stUserException2.etDiag														:= GD.ET_Diag.ExecutionAborted;
stUserException2.udiDiagExt													:= ET_DiagExt.Exception2FromVis;
stUserException2.sDiagExt													:= FC_EtDiagExtToString(ET_DiagExt.Exception2FromVis);
stUserException2.sMsg														:= 'Test Exception 2 from visualization - TPL.ET_Reaction.SyncStopEL';
stUserException2.udiModuleId												:= vpq_stMachineInterface.i_udiModuleId;
stUserException2.sModuleName												:= vpq_stMachineInterface.i_sModuleName;
stUserException2.etSource													:= TPL.ET_ExceptionSource.Vis;
stUserException2.timDelayTime												:= T#0MS;
stUserException2.wHmiAttributes												:= 0;
stUserException2.xAutoQuit													:= FALSE;
stUserException2.stReaction.axReaction[TPL.ET_Reaction.SyncStopEL]			:= TRUE;

stUserException3.etDiag														:= GD.ET_Diag.ExecutionAborted;
stUserException3.udiDiagExt													:= ET_DiagExt.Exception3FromVis;
stUserException3.sDiagExt													:= FC_EtDiagExtToString(ET_DiagExt.Exception3FromVis);
stUserException3.sMsg														:= 'Test Exception 3 from visualization - TPL.ET_Reaction.SyncStopEH';
stUserException3.udiModuleId												:= vpq_stMachineInterface.i_udiModuleId;
stUserException3.sModuleName												:= vpq_stMachineInterface.i_sModuleName;
stUserException3.etSource													:= TPL.ET_ExceptionSource.Vis;
stUserException3.timDelayTime												:= T#0MS;
stUserException3.wHmiAttributes												:= 0;
stUserException3.xAutoQuit													:= FALSE;
stUserException3.stReaction.axReaction[TPL.ET_Reaction.SyncStopEH]			:= TRUE;

stUserException4.etDiag														:= GD.ET_Diag.ExecutionAborted;
stUserException4.udiDiagExt													:= ET_DiagExt.Exception4FromVis;
stUserException4.sDiagExt													:= FC_EtDiagExtToString(ET_DiagExt.Exception4FromVis);
stUserException4.sMsg														:= 'Test Exception 4 from visualization - TPL.ET_Reaction.StopEndOfCycle';
stUserException4.udiModuleId												:= vpq_stMachineInterface.i_udiModuleId;
stUserException4.sModuleName												:= vpq_stMachineInterface.i_sModuleName;
stUserException4.etSource													:= TPL.ET_ExceptionSource.Vis;
stUserException4.timDelayTime												:= T#0MS;
stUserException4.wHmiAttributes												:= 0;
stUserException4.xAutoQuit													:= FALSE;
stUserException4.stReaction.axReaction[TPL.ET_Reaction.StopEndOfCycle]		:= TRUE;

stUserException5.etDiag														:= GD.ET_Diag.ExecutionAborted;
stUserException5.udiDiagExt													:= ET_DiagExt.Exception5FromVis;
stUserException5.sDiagExt													:= FC_EtDiagExtToString(ET_DiagExt.Exception5FromVis);
stUserException5.sMsg														:= 'Test Exception 5 from visualization - TPL.ET_Reaction.MainsContactorOff';
stUserException5.udiModuleId												:= vpq_stMachineInterface.i_udiModuleId;
stUserException5.sModuleName												:= vpq_stMachineInterface.i_sModuleName;
stUserException5.etSource													:= TPL.ET_ExceptionSource.Vis;
stUserException5.timDelayTime												:= T#0MS;
stUserException5.wHmiAttributes												:= 0;
stUserException5.xAutoQuit													:= FALSE;
stUserException5.stReaction.axReaction[TPL.ET_Reaction.MainsContactorOff]	:= TRUE;
stUserException5.stReaction.axReaction[TPL.ET_Reaction.StopEndOfCycle]		:= TRUE;
END_ACTION

ACTION LoggerVis:
(*For Displaying the LoggerList-Visualization Vis_Logger*)
IF vpiq_udiLogDataListIndexMin < 1 THEN
	vpiq_udiLogDataListIndexMin := 1;
END_IF

IF vpiq_udiLogDataListIndexMin > TPL.Gc_udiMaxNumberOfLogData - 11 THEN
	vpiq_udiLogDataListIndexMin := TPL.Gc_udiMaxNumberOfLogData - 11;
END_IF

FOR udiIndex2 := 1 TO 12 DO
	vpq_astLogDataTableAscii[udiIndex2] := G_stLogDataListAscii.astLogData[vpiq_udiLogDataListIndexMin + udiIndex2 - 1];

	IF G_stLogDataListAscii.astLogData[vpiq_udiLogDataListIndexMin + udiIndex2 - 1].asAsciiData[1]= 'Cmd come' THEN
			vpq_astLogDataTable[udiIndex2].etReason:= TPL. ET_LogDataFilter.CmdCome;
	ELSIF G_stLogDataListAscii.astLogData[vpiq_udiLogDataListIndexMin + udiIndex2 - 1].asAsciiData[1]= 'Cmd go' THEN
			vpq_astLogDataTable[udiIndex2].etReason:= TPL.ET_LogDataFilter.CmdGo;
	ELSIF G_stLogDataListAscii.astLogData[vpiq_udiLogDataListIndexMin + udiIndex2 - 1].asAsciiData[1]= 'StartStep come' THEN
			vpq_astLogDataTable[udiIndex2].etReason:= TPL.ET_LogDataFilter.StartStepCome;
	ELSIF G_stLogDataListAscii.astLogData[vpiq_udiLogDataListIndexMin + udiIndex2 - 1].asAsciiData[1]= 'StartStep go' THEN
			vpq_astLogDataTable[udiIndex2].etReason:= TPL.ET_LogDataFilter.StartStepGo;
	ELSIF G_stLogDataListAscii.astLogData[vpiq_udiLogDataListIndexMin + udiIndex2 - 1].asAsciiData[1]= 'Reaction come' THEN
			vpq_astLogDataTable[udiIndex2].etReason:= TPL.ET_LogDataFilter.ReactionCome;
	ELSIF G_stLogDataListAscii.astLogData[vpiq_udiLogDataListIndexMin + udiIndex2 - 1].asAsciiData[1]= 'Reaction go' THEN
			vpq_astLogDataTable[udiIndex2].etReason:= TPL.ET_LogDataFilter.ReactionGo;
	ELSIF G_stLogDataListAscii.astLogData[vpiq_udiLogDataListIndexMin + udiIndex2 - 1].asAsciiData[1]= 'Exception quit' THEN
			vpq_astLogDataTable[udiIndex2].etReason:= TPL.ET_LogDataFilter.ExceptionQuit;
	ELSIF G_stLogDataListAscii.astLogData[vpiq_udiLogDataListIndexMin + udiIndex2 - 1].asAsciiData[1]= 'Exception come' THEN
			vpq_astLogDataTable[udiIndex2].etReason := TPL.ET_LogDataFilter.ExceptionCome;
	ELSIF G_stLogDataListAscii.astLogData[vpiq_udiLogDataListIndexMin + udiIndex2 - 1].asAsciiData[1]= 'Exception autoquit' THEN
			vpq_astLogDataTable[udiIndex2].etReason:= TPL.ET_LogDataFilter.ExceptionAutoQuit;
	ELSIF G_stLogDataListAscii.astLogData[vpiq_udiLogDataListIndexMin + udiIndex2 - 1].asAsciiData[1]= 'User entry' THEN
			vpq_astLogDataTable[udiIndex2].etReason:= TPL.ET_LogDataFilter.User;
	ELSE
		vpq_astLogDataTable[udiIndex2].etReason:= TPL.ET_LogDataFilter.None;
	END_IF
	vpq_astLogDataTable[udiIndex2].dateDate 		:= STRING_TO_DATE(G_stLogDataListAscii.astLogData[vpiq_udiLogDataListIndexMin + udiIndex2 - 1].asAsciiData[2]);
	vpq_astLogDataTable[udiIndex2].todTime			:= STRING_TO_TOD(G_stLogDataListAscii.astLogData[vpiq_udiLogDataListIndexMin + udiIndex2 - 1].asAsciiData[3]);
	vpq_astLogDataTable[udiIndex2].udiModuleId		:= STRING_TO_UDINT(G_stLogDataListAscii.astLogData[vpiq_udiLogDataListIndexMin + udiIndex2 - 1].asAsciiData[4]);
	vpq_astLogDataTable[udiIndex2].sModuleName		:= G_stLogDataListAscii.astLogData[vpiq_udiLogDataListIndexMin + udiIndex2 - 1].asAsciiData[5];
	vpq_astLogDataTable[udiIndex2].diCMD			:= STRING_TO_DINT(G_stLogDataListAscii.astLogData[vpiq_udiLogDataListIndexMin + udiIndex2 - 1].asAsciiData[6]);
	vpq_astLogDataTable[udiIndex2].diStartStep		:= STRING_TO_DINT(G_stLogDataListAscii.astLogData[vpiq_udiLogDataListIndexMin + udiIndex2 - 1].asAsciiData[7]);

	vpq_astLogDataTable[udiIndex2].etDiag			:= STRING_TO_UDINT(G_stLogDataListAscii.astLogData[vpiq_udiLogDataListIndexMin + udiIndex2 - 1].asAsciiData[8]);
	vpq_astLogDataTable[udiIndex2].udiDiagExt		:= STRING_TO_UDINT(G_stLogDataListAscii.astLogData[vpiq_udiLogDataListIndexMin + udiIndex2 - 1].asAsciiData[10]);
	vpq_astLogDataTable[udiIndex2].sDiagExt			:= G_stLogDataListAscii.astLogData[vpiq_udiLogDataListIndexMin + udiIndex2 - 1].asAsciiData[11];
	vpq_astLogDataTable[udiIndex2].sMsg				:= G_stLogDataListAscii.astLogData[vpiq_udiLogDataListIndexMin + udiIndex2 - 1].asAsciiData[12];
	
	FOR udiIndex3 := 1 TO TPL.Gc_udiMaxNumberOfReactions DO
		IF FIND(G_stLogDataListAscii.astLogData[vpiq_udiLogDataListIndexMin + udiIndex2 - 1].asAsciiData[13], UDINT_TO_STRING(udiIndex3))<>0 THEN
			vpq_astLogDataTable[udiIndex2].stReaction.axReaction[udiIndex3] := TRUE;
		ELSE
			vpq_astLogDataTable[udiIndex2].stReaction.axReaction[udiIndex3] := FALSE;
		END_IF
	END_FOR

	IF    G_stLogDataListAscii.astLogData[vpiq_udiLogDataListIndexMin + udiIndex2 - 1].asAsciiData[14]= '1' THEN
		vpq_astLogDataTable[udiIndex2].etSource:= TPL.ET_ExceptionSource.ModuleController;
	ELSIF G_stLogDataListAscii.astLogData[vpiq_udiLogDataListIndexMin + udiIndex2 - 1].asAsciiData[14]= '2' THEN
		vpq_astLogDataTable[udiIndex2].etSource:= TPL.ET_ExceptionSource.ExceptionHandler;
	ELSIF G_stLogDataListAscii.astLogData[vpiq_udiLogDataListIndexMin + udiIndex2 - 1].asAsciiData[14]= '3' THEN
		vpq_astLogDataTable[udiIndex2].etSource:= TPL.ET_ExceptionSource.Logger;
	ELSIF G_stLogDataListAscii.astLogData[vpiq_udiLogDataListIndexMin + udiIndex2 - 1].asAsciiData[14]= '4' THEN
		vpq_astLogDataTable[udiIndex2].etSource:= TPL.ET_ExceptionSource.Main;
	ELSIF G_stLogDataListAscii.astLogData[vpiq_udiLogDataListIndexMin + udiIndex2 - 1].asAsciiData[14]= '5' THEN
		vpq_astLogDataTable[udiIndex2].etSource:= TPL.ET_ExceptionSource.Vis;
	ELSIF G_stLogDataListAscii.astLogData[vpiq_udiLogDataListIndexMin + udiIndex2 - 1].asAsciiData[14]= '6' THEN
		vpq_astLogDataTable[udiIndex2].etSource:= TPL.ET_ExceptionSource.User;
	ELSIF G_stLogDataListAscii.astLogData[vpiq_udiLogDataListIndexMin + udiIndex2 - 1].asAsciiData[14]= '7' THEN
		vpq_astLogDataTable[udiIndex2].etSource:= TPL.ET_ExceptionSource.NodeModule;
	ELSIF G_stLogDataListAscii.astLogData[vpiq_udiLogDataListIndexMin + udiIndex2 - 1].asAsciiData[14]= '8' THEN
		vpq_astLogDataTable[udiIndex2].etSource:= TPL.ET_ExceptionSource.AxisModule;
	ELSIF G_stLogDataListAscii.astLogData[vpiq_udiLogDataListIndexMin + udiIndex2 - 1].asAsciiData[14]= '9' THEN
		vpq_astLogDataTable[udiIndex2].etSource:= TPL.ET_ExceptionSource.MultiBeltModule;
	ELSIF G_stLogDataListAscii.astLogData[vpiq_udiLogDataListIndexMin + udiIndex2 - 1].asAsciiData[14]= '10' THEN
		vpq_astLogDataTable[udiIndex2].etSource:= TPL.ET_ExceptionSource.SmartInfeedModule;
	ELSIF G_stLogDataListAscii.astLogData[vpiq_udiLogDataListIndexMin + udiIndex2 - 1].asAsciiData[14]= '11' THEN
		vpq_astLogDataTable[udiIndex2].etSource:= TPL.ET_ExceptionSource.RoboticModule;
	ELSIF G_stLogDataListAscii.astLogData[vpiq_udiLogDataListIndexMin + udiIndex2 - 1].asAsciiData[14]= '12' THEN
		vpq_astLogDataTable[udiIndex2].etSource:= TPL.ET_ExceptionSource.UnwinderModule;
	ELSIF G_stLogDataListAscii.astLogData[vpiq_udiLogDataListIndexMin + udiIndex2 - 1].asAsciiData[14]= '13' THEN
		vpq_astLogDataTable[udiIndex2].etSource:= TPL.ET_ExceptionSource.SealingModule;
	ELSIF G_stLogDataListAscii.astLogData[vpiq_udiLogDataListIndexMin + udiIndex2 - 1].asAsciiData[14]= '14' THEN
		vpq_astLogDataTable[udiIndex2].etSource:= TPL.ET_ExceptionSource.AtvModule;
	ELSIF G_stLogDataListAscii.astLogData[vpiq_udiLogDataListIndexMin + udiIndex2 - 1].asAsciiData[14]= '15' THEN
		vpq_astLogDataTable[udiIndex2].etSource:= TPL.ET_ExceptionSource.IlxModule;
	ELSIF G_stLogDataListAscii.astLogData[vpiq_udiLogDataListIndexMin + udiIndex2 - 1].asAsciiData[14]= '16' THEN
		vpq_astLogDataTable[udiIndex2].etSource:= TPL.ET_ExceptionSource.CrankModule;
	ELSIF G_stLogDataListAscii.astLogData[vpiq_udiLogDataListIndexMin + udiIndex2 - 1].asAsciiData[14]= '17' THEN
		vpq_astLogDataTable[udiIndex2].etSource:= TPL.ET_ExceptionSource.ValveModule;
	ELSIF G_stLogDataListAscii.astLogData[vpiq_udiLogDataListIndexMin + udiIndex2 - 1].asAsciiData[14]= '18' THEN
		vpq_astLogDataTable[udiIndex2].etSource:= TPL.ET_ExceptionSource.CapperModule;
	ELSE
		vpq_astLogDataTable[udiIndex2].etSource:= TPL.ET_ExceptionSource.None;
	END_IF
	
	vpq_astLogDataTable[udiIndex2].xAutoQuit	:= STRING_TO_BOOL(G_stLogDataListAscii.astLogData[vpiq_udiLogDataListIndexMin + udiIndex2 - 1].asAsciiData[15]);
END_FOR


vpq_udiLogDataListIndexMax := vpiq_udiLogDataListIndexMin + 11;

vpiq_udiNumberOfLogData := G_stLogDataListAscii.udiNumberOfLogData;
IF vpq_udiLogDataListIndexMax > G_stLogDataListAscii.udiNumberOfLogData - 1  THEN
	vpq_xLogDataScrollDown := TRUE;

ELSE
	vpq_xLogDataScrollDown := FALSE;
END_IF

IF vpiq_xButtonLogDataListDetails AND NOT vpq_xShowLogDataListDetails THEN
	vpq_xShowLogDataListDetails				:= TRUE;
	vpiq_xButtonLogDataListDetails			:= FALSE;
ELSIF vpiq_xButtonLogDataListDetails AND vpq_xShowLogDataListDetails THEN
	vpq_xShowLogDataListDetails				:= FALSE;
	vpiq_xButtonLogDataListDetails			:= FALSE;
END_IF
END_ACTION

ACTION MainPageCmdTable:
(* Find the current table*)
vpq_udiNumberOfCmdStepsModule		:= 0; (* Default values, for security *)
pstEQCMDTableListEntry	:= 0;
pstEQCMDTable			:= 0;

IF(vpq_stMachineInterface.q_diCmdActive <> 0 AND vpq_stMachineInterface.iq_stExt.udiNumberOfCmdTables > 0 AND vpq_stMachineInterface.iq_stExt.pstListofCMDTables <> 0) THEN
	FOR udiTmp2 := 1 TO vpq_stMachineInterface.iq_stExt.udiNumberOfCMDTables DO
		pstEQCMDTableListEntry := vpq_stMachineInterface.iq_stExt.pstListofCMDTables +  UDINT_TO_DWORD((udiTmp2-1)*SIZEOF(pstEQCMDTableListEntry^));
		IF(pstEQCMDTableListEntry^.diCMD = vpq_stMachineInterface.q_diCmdActive) THEN (* Found *)
			vpq_udiNumberOfCmdStepsModule := pstEQCMDTableListEntry^.udiNumberOfCmdSteps;
			vpq_udiNumberOfCmdStepsMain := vpq_udiNumberOfCmdStepsModule;
			pstEQCMDTable := pstEQCMDTableListEntry^.pstCMDTable;
			vpq_sCmdTitelMain := pstEQCMDTableListEntry^.sTitle;
			EXIT;
		END_IF
	END_FOR
END_IF

(***********************************************************************************************************************)
(* Check the limits of the Vis/ shown table *)
udiIndexOldMainTable := 0;
IF vpiq_udiIndexMinMain <> udiIndexOldMainTable THEN
														(*More than 10 steps ??*)
	IF (vpiq_udiIndexMinMain + 9 < vpq_udiNumberOfCmdStepsMain) THEN
		udiIndexMaxMainTable := vpiq_udiIndexMinMain + 9;
	ELSE
		udiIndexMaxMainTable := vpq_udiNumberOfCmdStepsMain;
	END_IF
														(*Additional safety check*)
	IF (vpiq_udiIndexMinMain < 1) OR (vpiq_udiIndexMinMain > vpq_udiNumberOfCmdStepsMain) THEN
		vpiq_udiIndexMinMain :=1;
		udiIndexMaxMainTable := 10;
	END_IF

	udiIndexOldMainTable := vpiq_udiIndexMinMain;
END_IF (*udiEQMainTableIndexMin <> udiEQMainTableIndexOld*)

vpq_xDisableScrollUpMain	:= NOT (vpiq_udiIndexMinMain > 1);
vpq_xDisableScrollDownMain	:= NOT (vpiq_udiIndexMinMain + 9 < vpq_udiNumberOfCmdStepsMain) ;

(***********************************************************************************************************************)
(*Refresh the values in the table if more then "Max commands" should be shown!*)
IF(pstEQCMDTable <> 0) THEN
	FOR udiCounter := udiIndexOldMainTable TO udiIndexMaxMainTable DO
		pstEQCMDTableEntry := pstEQCMDTable +  UDINT_TO_DWORD(((udiCounter-1) * SIZEOF(pstEQCMDTable^)));
		vpq_astActualCmdTableMain[udiCounter - udiIndexOldMainTable + 1] := pstEQCMDTableEntry^;
	END_FOR
	FOR udiCounter := udiIndexMaxMainTable + 1 TO udiIndexOldMainTable + 9 DO
		vpq_astActualCmdTableMain[udiCounter - udiIndexOldMainTable + 1] := c_stEmptyCmdTableStep;
	END_FOR
END_IF
END_ACTION

ACTION ModuleNavigationIn:
(* Navigation *)

(* 2D navigation *)
IF(vpiq_xNavUp OR vpiq_xNavDown OR vpiq_xNavLeft OR vpiq_xNavRight) THEN
	IF vpiq_xNavRight THEN
		(* Move the the next module on the same level *)
		IF audiHierarchy[udiCurrentLevel] + 1 <= udiCurrentLevelSize + udiCurrentNumberOfControlModules  THEN
			audiHierarchy[udiCurrentLevel] := audiHierarchy[udiCurrentLevel] + 1;
			IF audiHierarchy[udiCurrentLevel]  > udiCurrentLevelSize THEN
				udiControlModuleSelectedInLevel	:= udiCurrentLevel;
				vpq_udiActiveControlModuleNumber:= audiHierarchy[udiCurrentLevel]-udiCurrentLevelSize;
			END_IF
		END_IF
	END_IF
	IF vpiq_xNavLeft THEN
		(* Move the the previous module on the same level *)
		IF audiHierarchy[udiCurrentLevel] -1 >= 1 THEN
			audiHierarchy[udiCurrentLevel] := audiHierarchy[udiCurrentLevel] - 1;
			vpq_udiActiveControlModuleNumber:= audiHierarchy[udiCurrentLevel]-udiCurrentLevelSize;
			IF audiHierarchy[udiCurrentLevel] <= udiCurrentLevelSize THEN
				udiControlModuleSelectedInLevel	:= 0;
				vpq_udiActiveControlModuleNumber:= 0;
			END_IF
		END_IF (* ELSE ignore *)
	END_IF
	IF vpiq_xNavUp THEN
		(* Move one level up *)
		udiControlModuleSelectedInLevel := 0;
		vpq_udiActiveControlModuleNumber:= 0;
		IF udiCurrentLevel - 1 >= 1 THEN
			udiCurrentLevel := udiCurrentLevel - 1;
		END_IF (* ELSE ignore *)
	END_IF
	IF vpiq_xNavDown THEN
		(* Move one level down *)
		IF (udiCurrentLevel + 1 <= c_udiMaxHierarchyLevels) AND (xCurrentHasSubModules OR xCurrentHasControlModules) THEN
			udiCurrentLevel := udiCurrentLevel + 1;
			audiHierarchy[udiCurrentLevel] := 1;
			IF NOT xCurrentHasSubModules AND xCurrentHasControlModules THEN
				udiControlModuleSelectedInLevel := udiCurrentLevel;
				vpq_udiActiveControlModuleNumber:= audiHierarchy[udiCurrentLevel];
			ELSE
				udiControlModuleSelectedInLevel	:= 0;
				vpq_udiActiveControlModuleNumber:= 0;
			END_IF

		END_IF (* ELSE ignore *)
	END_IF

	vpiq_xNavUp		:= FALSE;
	vpiq_xNavDown	:= FALSE;
	vpiq_xNavLeft	:= FALSE;
	vpiq_xNavRight	:= FALSE;
	
	xUpdateData := TRUE;
END_IF (* End 2D navbutton hit *)

(* Direct navigation (on level 2 and 3) *)
(* Module level *)
IF vpiq_axModuleList[1] OR vpiq_axModuleList[2] OR vpiq_axModuleList[3] OR vpiq_axModuleList[4] OR vpiq_axModuleList[5] OR
   vpiq_axControlModuleList[1] OR vpiq_axControlModuleList[2] OR vpiq_axControlModuleList[3] OR vpiq_axControlModuleList[4] OR vpiq_axControlModuleList[5] THEN
	udiCurrentLevel := 2;
	udiCurrentLevel := 2;
	FOR udiTmp := 1 TO 5 DO
		(*select an equipment module via the buttons on level 2*)
		IF(vpiq_axModuleList[udiTmp]) THEN
			audiHierarchy[udiCurrentLevel] := udiTmp + udiMinModuleList - 1;
			vpiq_axModuleList[udiTmp] := FALSE;
			udiControlModuleSelectedInLevel := 0;
			vpq_udiActiveControlModuleNumber:= 0;
		END_IF
		(*select a control module via the buttons on level 2*)
		IF vpiq_axControlModuleList[udiTmp] THEN
			audiHierarchy[udiCurrentLevel] := udiTmp + udiMinModuleList - 1;
			udiControlModuleSelectedInLevel	:= udiCurrentLevel;
			vpiq_axControlModuleList[udiTmp] := FALSE;
		END_IF
	END_FOR
	xUpdateData := TRUE;
END_IF
IF vpiq_xModuleListDown THEN
	vpiq_xModuleListDown := FALSE;
	IF(udiMinModuleList > 1) THEN
		udiMinModuleList := udiMinModuleList - 1;
	END_IF
	xUpdateData := TRUE;
END_IF
IF vpiq_xModuleListUp THEN
	vpiq_xModuleListUp := FALSE;
	IF(udiMinModuleList + 4 <= vpq_stMachineInterface.iq_stExt.udiNumberOfSubModules + vpq_stMachineInterface.iq_stExt.udiNumberOfControlModules) THEN
		udiMinModuleList := udiMinModuleList + 1;
	END_IF
	xUpdateData := TRUE;
END_IF
(* Submodule level *)
IF(udiCurrentLevel >= 2) THEN (* Impossible if the main machine is selected *)
	IF vpiq_axSubModuleList[1] OR vpiq_axSubModuleList[2] OR vpiq_axSubModuleList[3] OR vpiq_axSubModuleList[4] OR vpiq_axSubModuleList[5] OR
	   vpiq_axSubControlModuleList[1] OR vpiq_axSubControlModuleList[2] OR vpiq_axSubControlModuleList[3] OR vpiq_axSubControlModuleList[4] OR vpiq_axSubControlModuleList[5] THEN
		udiCurrentLevel := 3;
		FOR udiTmp := 1 TO 5 DO
			(*select an equipment module via the buttons on level 3*)
			IF(vpiq_axSubModuleList[udiTmp]) THEN
				audiHierarchy[udiCurrentLevel] := udiTmp + udiMinSubModuleList - 1;
				vpiq_axSubModuleList[udiTmp] := FALSE;
				udiControlModuleSelectedInLevel	:= 0;
				vpq_udiActiveControlModuleNumber	:= 0;
			END_IF
			(*select a control module via the buttons on level 3*)
			IF vpiq_axSubControlModuleList[udiTmp] THEN
				audiHierarchy[udiCurrentLevel] := udiTmp + udiMinSubModuleList - 1;
				vpiq_axSubControlModuleList[udiTmp] := FALSE;
				udiControlModuleSelectedInLevel	:= udiCurrentLevel;
			END_IF
		END_FOR
		xUpdateData := TRUE;
	END_IF
	IF vpiq_xSubModuleListDown THEN
		vpiq_xSubModuleListDown := FALSE;
		IF(udiMinSubModuleList > 1) THEN
			udiMinSubModuleList := udiMinSubModuleList - 1;
		END_IF
		xUpdateData := TRUE;
	END_IF
	IF vpiq_xSubModuleListUp THEN
		vpiq_xSubModuleListUp := FALSE;
		IF(udiMinSubModuleList + 4 < udiCurrentLevel3Size + udiNumberOfControlModulesLevel2) THEN
			udiMinSubModuleList := udiMinSubModuleList + 1;
		END_IF
		xUpdateData := TRUE;
	END_IF
END_IF
END_ACTION

ACTION ModuleNavigationOut:
(* update 2d nav data *)
vpq_sNameNavUp		:= '';
vpq_sNameNavRight	:= '';
vpq_sNameNavLeft		:= '';

IF pstCurrentParent = 0 THEN
	udiCurrentLevelSize := 1;
ELSE
	udiCurrentLevelSize := pstCurrentParent^.iq_stExt.udiNumberOfSubModules;

	vpq_sNameNavUp := pstCurrentParent^.i_sModuleName;
	(*If next module is a equipment module*)
	IF (audiHierarchy[udiCurrentLevel] + 1 <= udiCurrentLevelSize) THEN
		pstTmp := pstCurrentParent^.iq_stExt.dwSubModulesItf
			+ UDINT_TO_DWORD((audiHierarchy[udiCurrentLevel] -1 + 1) * SIZEOF(vpq_stCurrentModuleStandardInterface));
		vpq_sNameNavRight := pstTmp^.i_sModuleName;
	(*If next module is a control module*)
	ELSIF audiHierarchy[udiCurrentLevel] + 1 <= udiCurrentLevelSize + pstCurrentParent^.iq_stExt.udiNumberOfControlModules THEN
		pstControlModuleInterface	:= pstCurrentParent^.iq_stExt.dwControlModulesItf + UDINT_TO_DWORD((audiHierarchy[udiCurrentLevel]-udiCurrentLevelSize) * SIZEOF(pstControlModuleInterface^));
		vpq_sNameNavRight			:= pstControlModuleInterface^.sControlModuleName;
	END_IF
	IF (audiHierarchy[udiCurrentLevel] -1 >= 1) THEN
		(*If former module is a equipment module*)
		IF audiHierarchy[udiCurrentLevel]-1 <= udiCurrentLevelSize THEN
			pstTmp := pstCurrentParent^.iq_stExt.dwSubModulesItf
				+ UDINT_TO_DWORD((audiHierarchy[udiCurrentLevel] -1 - 1) * SIZEOF(vpq_stCurrentModuleStandardInterface));
			vpq_sNameNavLeft := pstTmp^.i_sModuleName;
		(*If former module is a control module*)
		ELSE
			pstControlModuleInterface	:= pstCurrentParent^.iq_stExt.dwControlModulesItf + UDINT_TO_DWORD((audiHierarchy[udiCurrentLevel]-udiCurrentLevelSize-2) * SIZEOF(pstControlModuleInterface^));
			vpq_sNameNavLeft				:= pstControlModuleInterface^.sControlModuleName;
		END_IF
	END_IF
END_IF

xCurrentHasControlModules := pstCurrent^.iq_stExt.udiNumberOfControlModules > 0;
xCurrentHasSubModules := ((pstCurrent^.iq_stExt.udiNumberOfSubModules > 0) AND udiControlModuleSelectedInLevel = 0);
xCurrentIsNoNodeModule := (pstCurrent^.q_dwModuleType <>  UDINT_TO_DWORD(TPL.ET_ModuleType.NodeModule));
IF((xCurrentIsNoNodeModule OR xCurrentHasControlModules) AND udiControlModuleSelectedInLevel = 0) THEN
	IF(pstCurrentParent <> 0) THEN (* Security check *)
		pdwTmp := ADR(pstCurrentParent^.iq_stExt.pdwSubModulesAddItf^)
			+  UDINT_TO_DWORD((audiHierarchy[udiCurrentLevel] - 1) * SIZEOF(dwDummy));
		dwCurrentAddInterface := pdwTmp^;
	END_IF
END_IF

vpq_xEnableNavUp		:= (udiCurrentLevel - 1 >= 1);
vpq_xEnableNavDown	:= (udiCurrentLevel < c_udiMaxHierarchyLevels) AND (xCurrentHasSubModules OR xCurrentHasControlModules) AND udiControlModuleSelectedInLevel = 0 ;
vpq_xEnableNavLeft	:= (audiHierarchy[udiCurrentLevel] -1 >= 1);
vpq_xEnableNavRight	:= (audiHierarchy[udiCurrentLevel] + 1 <= udiCurrentLevelSize + udiCurrentNumberOfControlModules)AND(udiCurrentLevel >=2);

IF vpq_xEnableNavDown THEN
	(* Name of the first submodule of the current module *)
	IF xCurrentHasSubModules THEN
		pstTmp := pstCurrent^.iq_stExt.dwSubModulesItf;
		vpq_sNameNavDown := pstTmp^.i_sModuleName;
	ELSE
		pstControlModuleInterface	:= pstCurrent^.iq_stExt.dwControlModulesItf;
		vpq_sNameNavDown				:= pstControlModuleInterface^.sControlModuleName;
	END_IF

ELSE
	vpq_sNameNavDown := '';
END_IF

(* Update direct nav data *)
(* Module level *)
vpq_xDisableModuleListDown	:= NOT (udiMinModuleList > 1);
vpq_xDisableModuleListUp		:= NOT (udiMinModuleList + 5 <= vpq_stMachineInterface.iq_stExt.udiNumberOfSubModules + vpq_stMachineInterface.iq_stExt.udiNumberOfControlModules);
FOR udiTmp := 1 TO 5 DO
	vpq_axControlModuleValid[udiTmp]:=FALSE;
	audiControlModuleNumber[udiTmp]:= 0 (*-1*);
	vpq_asToolTipControlModuleList[udiTmp] := 'None';
	vpq_axDisableModuleList[udiTmp] := NOT ((udiTmp - 1 + udiMinModuleList) <= vpq_stMachineInterface.iq_stExt.udiNumberOfSubModules);
	vpq_axActiveModuleList[udiTmp] := (udiCurrentLevel >= 2) AND (audiHierarchy[2] = (udiTmp - 1 + udiMinModuleList));
	vpq_axControlModuleActive[udiTmp] := FALSE;
	(*Show button for equipment module*)
	IF(NOT vpq_axDisableModuleList[udiTmp]) THEN
		pstTmp := vpq_stMachineInterface.iq_stExt.dwSubModulesItf
			+ UDINT_TO_DWORD(((udiTmp - 1 + udiMinModuleList) - 1) * SIZEOF(vpq_stCurrentModuleStandardInterface));
		vpq_audiIdModuleList[udiTmp] := pstTmp^.i_udiModuleId;
		vpq_axIdModuleListValid[udiTmp] := TRUE;
		
		vpq_asNameModuleList[udiTmp] := pstTmp^.i_sModuleName;
	(*Show button for control module*)
	ELSE
		vpq_audiIdModuleList[udiTmp] := 0 (*-1*);
		vpq_axIdModuleListValid[udiTmp] := FALSE;
		vpq_asNameModuleList[udiTmp] := 'None';
		IF vpq_stMachineInterface.iq_stExt.udiNumberOfControlModules <> 0 AND udiTmp <= vpq_stMachineInterface.iq_stExt.udiNumberOfControlModules + vpq_stMachineInterface.iq_stExt.udiNumberOfSubModules THEN
			pstControlModuleInterface	:= vpq_stMachineInterface.iq_stExt.dwControlModulesItf + UDINT_TO_DWORD((udiTmp - vpq_stMachineInterface.iq_stExt.udiNumberOfSubModules - 1 + udiMinModuleList)-1) * SIZEOF(pstControlModuleInterface^);
			vpq_asToolTipControlModuleList[udiTmp]:= pstControlModuleInterface^.sControlModuleName;
			vpq_axControlModuleActive[udiTmp] := (udiCurrentLevel >= 2) AND (audiHierarchy[2] = (udiTmp - 1 + udiMinModuleList));
			vpq_axControlModuleValid[udiTmp]:=TRUE;
			audiControlModuleNumber[udiTmp]:= pstControlModuleInterface^.udiControlModuleNumber;
			vpq_asControlModuleButtonName[udiTmp]:= CONCAT(STR1:='Type: ',STR2:= CONCAT(STR1:= UDINT_TO_STRING(pstControlModuleInterface^.udiControlModuleType), STR2:= CONCAT(STR1:='   #: ',STR2:= UDINT_TO_STRING(pstControlModuleInterface^.udiControlModuleNumber))));
		END_IF
	END_IF
END_FOR

(* Submodule level *)
IF (udiMinSubModuleList + 4 > udiCurrentLevel3Size+udiNumberOfControlModulesLevel2) THEN
	udiMinSubModuleList := 1;
END_IF
vpq_xDisableSubModuleListDown	:= NOT (udiMinSubModuleList > 1);
vpq_xDisableSubModuleListUp		:= NOT (udiMinSubModuleList + 5 <= udiCurrentLevel3Size+udiNumberOfControlModulesLevel2)AND NOT (udiCurrentLevel = 2 AND xControlModuleSelected);
FOR udiTmp := 1 TO 5 DO
	vpq_axDisableSubModuleList[udiTmp] := NOT ((udiTmp - 1 + udiMinSubModuleList) <= udiCurrentLevel3Size);
	vpq_axActiveSubModuleList[udiTmp] := (udiCurrentLevel >= 3) AND (audiHierarchy[3] = (udiTmp - 1 + udiMinSubModuleList));
	vpq_audiIdSubModuleList[udiTmp] := 0 (*-1*);
	vpq_axIdSubModuleListValid[udiTmp] := FALSE;
	vpq_asNameSubModuleList[udiTmp] := 'None';
	vpq_axSubControlModuleValid[udiTmp]:= FALSE;
	audiSubControlModuleID[udiTmp]:= 0 (*-1*);
	vpq_asToolTipSubControlModuleList[udiTmp] := 'None';
	vpq_axSubControlModuleActive[udiTmp] := FALSE;
	(*Show button for equipment module*)
	IF(NOT vpq_axDisableSubModuleList[udiTmp]) THEN
		IF(pstCurrentFirstLevel3Module <> 0) THEN
			pstTmp := ADR(pstCurrentFirstLevel3Module^)
				+  UDINT_TO_DWORD(((udiTmp - 1 + udiMinSubModuleList) - 1) * SIZEOF(vpq_stCurrentModuleStandardInterface));
			vpq_audiIdSubModuleList[udiTmp] := pstTmp^.i_udiModuleId;
			vpq_axIdSubModuleListValid[udiTmp] := TRUE;
			
			vpq_asNameSubModuleList[udiTmp] := pstTmp^.i_sModuleName;
		END_IF
	(*Show button for control module*)
	ELSE
		IF udiCurrentLevel >= 2 AND udiControlModuleSelectedInLevel <> 2 THEN
			IF pstCurrentLevel2 <> 0 THEN
				IF pstCurrentLevel2^.iq_stExt.udiNumberOfControlModules <> 0 AND udiTmp <= pstCurrentLevel2^.iq_stExt.udiNumberOfControlModules + udiCurrentLevel3Size THEN
					pstControlModuleInterface	:= pstCurrentLevel2^.iq_stExt.dwControlModulesItf + UDINT_TO_DWORD((udiTmp - pstCurrentLevel2^.iq_stExt.udiNumberOfSubModules - 1 + udiMinSubModuleList - 1) * SIZEOF(pstControlModuleInterface^));
					vpq_asToolTipSubControlModuleList[udiTmp]:= pstControlModuleInterface^.sControlModuleName;
					vpq_asSubControlModuleButtonName[udiTmp]:= CONCAT(STR1:='Type: ',STR2:= CONCAT(STR1:= UDINT_TO_STRING(pstControlModuleInterface^.udiControlModuleType), STR2:= CONCAT(STR1:='   #: ',STR2:= UDINT_TO_STRING(pstControlModuleInterface^.udiControlModuleNumber))));
					vpq_axSubControlModuleActive[udiTmp] :=  (udiCurrentLevel >= 3) AND (audiHierarchy[3] = (udiTmp - 1 + udiMinSubModuleList));
					vpq_axSubControlModuleValid[udiTmp]:= TRUE;
					audiSubControlModuleID[udiTmp]:= pstControlModuleInterface^.udiControlModuleNumber;
				END_IF
			END_IF
		END_IF
	END_IF
END_FOR

// iEQTableIndexMin := 1;
//iEQTableIndexOld := 0;

(*Select current control module*)
FOR udiTmp := 1 TO 5 DO
	IF vpq_axControlModuleActive[udiTmp] THEN
		vpq_udiActiveControlModuleNumber:= audiControlModuleNumber[udiTmp];
	END_IF
	IF vpq_axSubControlModuleActive[udiTmp] THEN
		vpq_udiActiveControlModuleNumber:= audiSubControlModuleID[udiTmp];
	END_IF
END_FOR
END_ACTION

ACTION ModuleReaction:
stModuleReactions		:=pstCurrent^.i_stReaction;

IF vpiq_xModuleReactionUp THEN
	vpq_udiModuleReactionIndexMin := vpq_udiModuleReactionIndexMin + 1;
	vpiq_xModuleReactionUp := FALSE;
ELSIF vpiq_xModuleReactionDown THEN
	vpq_udiModuleReactionIndexMin := vpq_udiModuleReactionIndexMin - 1;
	vpiq_xModuleReactionDown := FALSE;
END_IF

IF vpq_udiModuleReactionIndexMin <> udiModuleReactionIndexOld THEN
														(*More than 10 steps ??*)
	IF (vpq_udiModuleReactionIndexMin + 9 < TPL.Gc_udiMaxNumberOfReactions) THEN
		udiModuleReactionIndexMax := vpq_udiModuleReactionIndexMin + 9;
	ELSE
		udiModuleReactionIndexMax := TPL.Gc_udiMaxNumberOfReactions;
	END_IF
														(*Additional safety check*)
	IF (vpq_udiModuleReactionIndexMin < 1) THEN
		vpq_udiModuleReactionIndexMin :=1;
		udiModuleReactionIndexMax := 10;
 	ELSIF (vpq_udiModuleReactionIndexMin > TPL.Gc_udiMaxNumberOfReactions-9)THEN
		vpq_udiModuleReactionIndexMin :=TPL.Gc_udiMaxNumberOfReactions-9;
		udiModuleReactionIndexMax := 10;
	END_IF

	udiModuleReactionIndexOld := vpq_udiModuleReactionIndexMin;
END_IF

IF TPL.Gc_udiMaxNumberOfReactions<10 THEN
	udiMaxValue := TPL.Gc_udiMaxNumberOfReactions;
ELSE
	udiMaxValue := 10;
END_IF

FOR udiCount2 := 1 TO udiMaxValue  DO
	vpq_axModuleReaction[udiCount2] := stModuleReactions.axReaction[vpq_udiModuleReactionIndexMin + udiCount2 - 1];
END_FOR
END_ACTION

ACTION ModuleVisController:
(* Begin of area for vis control fbs of different module types *)
(* SetCurrentModule(); has to be called after each special vis-controller, because it could have requested to change the current module via diSetAsCurrentModule *)

vpiq_fbAxisModuleVisController(	i_xEnable				:= vpq_xDoEnable, 
								i_pstMachineStandardItf	:= ADR(SR_MainMachine.stMachineInterface),
								i_pstCurrentStandardItf	:= pstCurrent, 
								i_dwCurrentAddItf		:= dwCurrentAddInterface, 
								i_xUpdateData			:= xUpdateForOtherFBs,
								i_udiCurrentJogTarget	:= G_udiManualModuleSelect, 
								iq_stExceptionList		:= G_stExceptionList,
								iq_stLogDataList		:= G_stLogDataList,
								q_xActive				=> , 
								q_xReady				=> , 
								q_etDiag				=> , 
								q_etDiagExt				=> , 
								q_sMsg					=> , 
								q_udiSetAsCurrentModule	=> udiSetAsCurrentModule,
								q_udiSetAsJogTarget		=> udiSetAsJogTarget);
SetCurrentModule();

(* Example 
vpiq_fbExampleLeafModuleVisController(	i_xEnable				:= vpq_xDoEnable, 
										i_pstMachineStandardItf	:= ADR(SR_MainMachine.stMachineInterface), 
										i_pstCurrentStandardItf	:= pstCurrent, 
										i_dwCurrentAddItf		:= dwCurrentAddInterface, 
										i_xUpdateData			:= xUpdateForOtherFBs, 
										i_udiCurrentJogTarget	:= G_udiManualModuleSelect, 
										iq_stExceptionList		:= G_stExceptionList,
										iq_stLogDataList		:= G_stLogDataList, 
										q_xActive				=> , 
										q_xReady				=> , 
										q_etDiag				=> , 
										q_etDiagExt				=> , 
										q_sMsg					=> , 
										q_udiSetAsCurrentModule	=> udiSetAsCurrentModule, 
										q_udiSetAsJogTarget		=> udiSetAsJogTarget);
SetCurrentModule();
*)

(* RoboticModule *)
(*vpiq_fbRoboticModuleVisController(	i_xEnable				:= vpq_xDoEnable, 
									i_pstMachineStandardItf	:= ADR(SR_MainMachine.stMachineInterface),
									i_pstCurrentStandardItf	:= pstCurrent, 
									i_dwCurrentAddItf		:= dwCurrentAddInterface, 
									i_xUpdateData			:= xUpdateForOtherFBs,
									i_udiCurrentJogTarget	:= G_udiManualModuleSelect, 
									iq_stExceptionList		:= G_stExceptionList,
									iq_stLogDataList		:= G_stLogDataList,
									q_xActive				=> , 
									q_xReady				=> , 
									q_etDiag				=> , 
									q_etDiagExt				=> , 
									q_sMsg					=> , 
									q_udiSetAsCurrentModule	=> udiSetAsCurrentModule,
									q_udiSetAsJogTarget		=> udiSetAsJogTarget);
SetCurrentModule();*)
END_ACTION

ACTION OpModeControl:
IFB_RTOPMode(CLK:= G_xDoPrepare OR G_xDoAuto OR G_xDoManual OR G_xDoJogMachine OR G_xDoBrakeRelease OR G_xDoTestMulticarrier OR G_xDoTrackCalibration);
IF G_xDoPrepare THEN
	IF g_xPrepareActive AND G_xPrepareEpas AND IFB_RTOPMode.Q THEN
		g_xPrepareActive := FALSE;
		G_xPrepareEpas:= FALSE;
	ELSIF IFB_RTOPMode.Q THEN
		g_xPrepareActive := TRUE;
		G_xPrepareEpas:= TRUE;
	END_IF
	G_xTestMulticarrierEpas := FALSE;
	G_xAutoEpas := FALSE;
	G_xManualEpas := FALSE;
	G_xJogMachineEpas := FALSE;
	G_xBrakeReleaseEpas := FALSE;
	G_xTrackCalibrationEpas := FALSE;

ELSIF G_xDoAuto THEN
	IF G_xAutoActive AND G_xAutoEpas AND IFB_RTOPMode.Q THEN
		G_xAutoActive := FALSE;
		G_xAutoEpas := FALSE;
	ELSIF IFB_RTOPMode.Q THEN
		G_xAutoActive := TRUE;
		G_xAutoEpas := TRUE;
	END_IF
	G_xTestMulticarrierEpas := FALSE;
	G_xManualEpas := FALSE;
	G_xJogMachineEpas := FALSE;
	G_xBrakeReleaseEpas := FALSE;
	G_xPrepareEpas:= FALSE;
	G_xTrackCalibrationEpas := FALSE;

ELSIF G_xDoManual THEN
	IF G_xManualActive AND G_xManualEpas AND IFB_RTOPMode.Q THEN
		G_xManualActive := FALSE;
		G_xManualEpas := FALSE;
	ELSIF IFB_RTOPMode.Q THEN
		g_xManualActive := TRUE;
		G_xManualEpas := TRUE;
	END_IF
	G_xTestMulticarrierEpas := FALSE;
	G_xJogMachineEpas := FALSE;
	G_xBrakeReleaseEpas := FALSE;
	G_xPrepareEpas:= FALSE;
	G_xAutoEpas := FALSE;
	G_xTrackCalibrationEpas := FALSE;

ELSIF g_xDoJogMachine THEN
	IF g_xJogMachineActive AND G_xJogMachineEpas AND IFB_RTOPMode.Q THEN
		g_xJogMachineActive := FALSE;
		G_xJogMachineEpas := FALSE;
	ELSIF IFB_RTOPMode.Q THEN
		g_xJogMachineActive := TRUE;
		G_xJogMachineEpas := TRUE;
	END_IF
	G_xTestMulticarrierEpas := FALSE;
	G_xBrakeReleaseEpas := FALSE;
	G_xPrepareEpas:= FALSE;
	G_xAutoEpas := FALSE;
	G_xManualEpas := FALSE;
	G_xTrackCalibrationEpas := FALSE;

ELSIF g_xDoBrakeRelease THEN
	IF g_xBrakeReleaseActive AND G_xBrakeReleaseEpas AND IFB_RTOPMode.Q THEN
		g_xBrakeReleaseActive := FALSE;
		G_xBrakeReleaseEpas := FALSE;
	ELSIF IFB_RTOPMode.Q THEN
		g_xBrakeReleaseActive := TRUE;
		G_xBrakeReleaseEpas := TRUE;
	END_IF
	G_xTestMulticarrierEpas := FALSE;
	G_xPrepareEpas:= FALSE;
	G_xAutoEpas := FALSE;
	G_xManualEpas := FALSE;
	G_xJogMachineEpas := FALSE;
	G_xTrackCalibrationEpas := FALSE;

ELSIF G_xDoTestMulticarrier THEN
	IF G_xTestMulticarrierActive AND G_xTestMulticarrierEpas AND IFB_RTOPMode.Q THEN
		G_xTestMulticarrierActive := FALSE;
		G_xTestMulticarrierEpas := FALSE;
	ELSIF IFB_RTOPMode.Q THEN
		G_xTestMulticarrierActive := TRUE;
		G_xTestMulticarrierEpas := TRUE;
	END_IF
	G_xBrakeReleaseEpas := FALSE;
	G_xPrepareEpas:= FALSE;
	G_xAutoEpas := FALSE;
	G_xManualEpas := FALSE;
	G_xJogMachineEpas := FALSE;
	G_xTrackCalibrationEpas := FALSE;
	
ELSIF G_xDoTrackCalibration THEN
	IF G_xTrackCalibrationActive AND G_xTrackCalibrationEpas AND IFB_RTOPMode.Q THEN
		G_xTrackCalibrationActive := FALSE;
		G_xTrackCalibrationEpas := FALSE;
	ELSIF IFB_RTOPMode.Q THEN
		G_xTrackCalibrationActive := TRUE;
		G_xTrackCalibrationEpas := TRUE;
	END_IF
	G_xTestMulticarrierEpas := FALSE;
	G_xBrakeReleaseEpas := FALSE;
	G_xPrepareEpas:= FALSE;
	G_xAutoEpas := FALSE;
	G_xManualEpas := FALSE;
	G_xJogMachineEpas := FALSE;
END_IF

IF g_xDoPrepare OR  g_xDoAuto OR g_xDoManual OR g_xDoJogMachine OR g_xDoBrakeRelease OR G_xDoTestMulticarrier OR G_xDoTrackCalibration THEN
	g_xPrepareActive := g_xPrepareActive  AND NOT( g_xDoAuto OR g_xDoManual OR g_xDoJogMachine OR g_xDoBrakeRelease  OR G_xDoTestMulticarrier OR G_xDoTrackCalibration);
	g_xAutoActive :=  g_xAutoActive AND NOT( g_xDoPrepare OR g_xDoManual OR g_xDoJogMachine OR g_xDoBrakeRelease OR G_xDoTestMulticarrier OR G_xDoTrackCalibration);
	g_xManualActive := g_xManualActive AND NOT( g_xDoPrepare OR g_xDoAuto OR g_xDoJogMachine OR g_xDoBrakeRelease OR G_xDoTestMulticarrier OR G_xDoTrackCalibration);
	g_xJogMachineActive :=  g_xJogMachineActive AND NOT( g_xDoPrepare OR g_xDoAuto OR g_xDoManual OR g_xDoBrakeRelease OR G_xDoTestMulticarrier OR G_xDoTrackCalibration);
	g_xBrakeReleaseActive:=  g_xBrakeReleaseActive  AND NOT( g_xDoPrepare OR g_xDoAuto OR g_xDoManual OR g_xDoJogMachine OR G_xDoTestMulticarrier OR G_xDoTrackCalibration);
	G_xTestMulticarrierActive:=  G_xTestMulticarrierActive  AND NOT( g_xDoPrepare OR g_xDoAuto OR g_xDoManual OR g_xDoJogMachine OR g_xDoBrakeRelease OR G_xDoTrackCalibration);
	G_xTrackCalibrationActive:=  G_xTrackCalibrationActive  AND NOT( g_xDoPrepare OR g_xDoAuto OR g_xDoManual OR g_xDoJogMachine OR g_xDoBrakeRelease OR G_xDoTestMulticarrier);
END_IF
END_ACTION

ACTION SearchCurrentModule:
(* Locate the current module according to the information in audiHierarchy *)
udiCurrentLevel3Size := 0;
pstCurrentFirstLevel3Module := 0;
pstCurrentParent := 0;
dwCurrentAddInterface := 0;
pstCurrent := ADR(SR_MainMachine.stMachineInterface); (* here we have to start at SR_MainMachine.stMachineInterface
instead of our local copy because otherwise it would not be possible to send commands to the MainMachine using the Vis. *)
FOR udiTmp := 2 TO udiCurrentLevel DO
	(* Only navigate to existing modules *)
	IF(pstCurrent^.iq_stExt.udiNumberOfSubModules + pstCurrent^.iq_stExt.udiNumberOfControlModules < audiHierarchy[udiTmp]) THEN
		audiHierarchy[udiTmp] := pstCurrent^.iq_stExt.udiNumberOfSubModules + pstCurrent^.iq_stExt.udiNumberOfControlModules;
	END_IF
	IF(audiHierarchy[udiTmp] <= 0) THEN
		audiHierarchy[udiTmp] := 1;
	END_IF
	IF(pstCurrent^.iq_stExt.udiNumberOfSubModules = 0 AND pstCurrent^.iq_stExt.udiNumberOfControlModules = 0) THEN
		(* Stop, the hierarchy was invalid *)
		udiCurrentLevel := udiTmp - 1;
	ELSE
		(* In case the stSubModules structure of this module is invalid, create an error and stop *)
		IF(pstCurrent^.iq_stExt.dwSubModulesItf = 0) THEN
			stPointerException.sMsg:=						'SR_VisControl: dwSubModuleInterfaces of module was 0';
		END_IF
		IF (pstCurrent^.iq_stExt.pdwSubModulesAddItf = 0 AND pstCurrent^.iq_stExt.dwControlModulesItf = 0) THEN
			stPointerException.sMsg:=						'SR_VisControl: pdwSubModuleAddInterfaces of module was 0';
		END_IF
		(*Set an error if there is no sub module (control module or equipment module)*)
		IF( (pstCurrent^.iq_stExt.dwSubModulesItf = 0 )
			OR (pstCurrent^.iq_stExt.pdwSubModulesAddItf = 0) ) AND pstCurrent^.iq_stExt.dwControlModulesItf = 0 THEN
			(* Error, the structures are not set in the expected way *)
		
			stPointerException.etDiag			:= GD.ET_Diag.UnexpectedProgramBehavior;
			stPointerException.udiDiagExt		:= ET_DiagExt.InvalidPointer;
			stPointerException.sDiagExt			:= FC_EtDiagExtToString(stPointerException.udiDiagExt);
//			stPointerException.sMsg				:= '';
			stPointerException.udiModuleId		:= pstCurrent^.i_udiModuleId;
			stPointerException.sModuleName		:= pstCurrent^.i_sModuleName;
			stPointerException.etSource			:= TPL.ET_ExceptionSource.Vis;
			stPointerException.timDelayTime		:= T#0MS;
			stPointerException.wHmiAttributes	:= 0;
			stPointerException.xAutoQuit		:= FALSE;
			stPointerException.stReaction.axReaction[TPL.ET_Reaction.AsyncStop] := TRUE;

			TPL.FC_SetException(i_xExceptionActive	:= TRUE,
								iq_stException		:= stPointerException,
								iq_stExceptionList	:= G_stExceptionList,
								iq_stLogDataList	:= G_stLogDataList);
								
			xPointerExceptionActive := TRUE;
			RETURN;
		END_IF
		
		pstCurrentParent := pstCurrent;
		(* Only navigate to existing equipment modules *)
		IF pstCurrentParent^.iq_stExt.udiNumberOfSubModules >= audiHierarchy[udiTmp] THEN
			pstCurrent := pstCurrent^.iq_stExt.dwSubModulesItf
				+ UDINT_TO_DWORD((audiHierarchy[udiTmp] - 1) * SIZEOF(vpq_stCurrentModuleStandardInterface));
			IF(udiTmp = 2) THEN
				udiCurrentLevel3Size := pstCurrent^.iq_stExt.udiNumberOfSubModules;
				pstCurrentFirstLevel3Module := pstCurrent^.iq_stExt.dwSubModulesItf;
			END_IF
		END_IF
		(*Initialize pointer for level 2*)
		IF udiTmp = 2 THEN
			pstCurrentLevel2 := pstCurrent;
		END_IF

	END_IF
END_FOR

(*Set pointer to the current module interface*)
IF pstCurrentParent = 0  THEN
	pstCurrentControlModuleStandardInterface 	:= pstCurrent^.iq_stExt.dwControlModulesItf;
	udiCurrentNumberOfControlModules 			:= pstCurrent^.iq_stExt.udiNumberOfControlModules;
ELSE
	pstCurrentControlModuleStandardInterface 	:= pstCurrentParent^.iq_stExt.dwControlModulesItf;
	udiCurrentNumberOfControlModules 			:= pstCurrentParent^.iq_stExt.udiNumberOfControlModules;
END_IF
IF pstCurrentLevel2 <> 0 THEN
	udiNumberOfControlModulesLevel2:= pstCurrentLevel2^.iq_stExt.udiNumberOfControlModules;
ELSE
	udiNumberOfControlModulesLevel2:= 0;
END_IF
END_ACTION

ACTION SetCurrentModule:
(*
	handles all requests coming from the special vis controllers

	sets the current module by modifying aiHierachy
	also sets the jog target

inputs:
	diSetAsCurrentModule - if <> 0 contains the module ID of the module to set as current module

in_out:
	audiHierarchy	
	udiCurrentLevel

flags:
	

*)
IF(udiSetAsCurrentModule > 0) THEN
	udiTmp2 := 1;
	WHILE(udiSetAsCurrentModule > udiTmp2 * 100) DO
		udiTmp2 := udiTmp2 * 100;
	END_WHILE

	udiCurrentLevel := 0;
	WHILE(udiTmp2 > 0) DO
		udiCurrentLevel := udiCurrentLevel + 1;
		audiHierarchy[udiCurrentLevel] := udiSetAsCurrentModule / udiTmp2;
		udiSetAsCurrentModule := udiSetAsCurrentModule MOD udiTmp2;
		udiTmp2 := udiTmp2 / 100;
	END_WHILE

	IF(udiCurrentLevel < 1) THEN
		udiCurrentLevel := 1;
	END_IF

	udiSetAsCurrentModule := 0;
	xUpdateData := TRUE;
END_IF

IF(udiSetAsJogTarget <> 0) THEN
	G_udiManualModuleSelect		:= udiSetAsJogTarget;
//	G_udiManualElementSelect	:= udiSetAsJogTargetNum;
	udiSetAsJogTarget := 0;
//	udiSetAsJogTargetNum := 0;
END_IF
END_ACTION

END_PROGRAM

// LMC_PacDrive/Application/TemplateFullProgrammingFramework/Examples/ExampleLeafModule/FB_ExampleLeafModuleVisController
FUNCTION_BLOCK FB_ExampleLeafModuleVisController

VAR_INPUT
	i_xEnable								: BOOL;
	i_pstMachineStandardItf					: POINTER TO TPL.ST_StandardModuleInterface;
	i_pstCurrentStandardItf					: POINTER TO TPL.ST_StandardModuleInterface;
	i_dwCurrentAddItf						: DWORD;
	i_xUpdateData							: BOOL; (* Signals the selection of another module *)
	i_udiCurrentJogTarget					: UDINT;
END_VAR

VAR_IN_OUT
	iq_stExceptionList				: TPL.ST_ExceptionList;
	iq_stLogDataList	   			: TPL.ST_LogDataList;
END_VAR

VAR_OUTPUT
	q_xActive								: BOOL;
	q_xReady								: BOOL;
	q_etDiag								: GD.ET_Diag := GD.ET_Diag.Ok;
	q_etDiagExt								: ET_DiagExtExampleLeafModule := ET_DiagExtExampleLeafModule.Disabled;
	q_sMsg									: STRING[80] := '';
	q_udiSetAsCurrentModule					: UDINT; (* A moduleID, if <> 0, it is set as the current module *)
	q_udiSetAsJogTarget						: UDINT;
END_VAR

VAR
	xCurrentIsOfMyType						: BOOL;
	pstCurrentExampleLeafModuleInterface	: POINTER TO ST_ExampleLeafModuleInterface;
	stCurrentExampleLeafModuleInterface		: ST_ExampleLeafModuleInterface;
	iPaneSelect								: INT := 1; (* Variable for selecting the active pane *)

	(* Variables to detect user changes in the vis *)
	xInitUserInputs							: BOOL;

	(* list of all example leaf modules in the machine *)
	audiExampleLeafModuleId					: ARRAY[1..c_udiMaxExampleLeafModules] OF UDINT; (* if <> 0, module exists *)
	asExampleLeafModuleName					: ARRAY[1..c_udiMaxExampleLeafModules] OF STRING[80]; (* if <> 0, module exists *)
	udiCountExampleLeafModules				: UDINT;
	udiSetAsCurrentModule					: UDINT;

	(* temporary variable, not to be used after init *)
	apExampleLeafModuleInterface			: ARRAY[1..c_udiMaxExampleLeafModules] OF POINTER TO TPL.ST_StandardModuleInterface;
	udiTmp									: UDINT;
	xEnableFlag								: BOOL;

	(* Variables to detect user changes in the vis *)
	lrPosMax								: LREAL;
END_VAR

VAR CONSTANT
	c_udiMaxExampleLeafModules : UDINT := 10;
END_VAR

q_udiSetAsCurrentModule 	:= 0;
q_udiSetAsJogTarget			:= 0;

(*********************************************************************)

IF i_xEnable AND NOT xEnableFlag THEN
	xEnableFlag := TRUE;
	
	q_xActive	:= TRUE;	
	
	q_etDiag	:= GD.ET_Diag.Ok;
	q_etDiagExt := ET_DiagExtExampleLeafModule.Initializing;
	q_sMsg		:= '';
	
	
		
	udiCountExampleLeafModules := TPL.FC_GetAllModulesOfType(	i_pstMachineStandardItf	:= i_pstMachineStandardItf,
																i_dwWantedType			:= ET_ModuleType.ExampleLeafModule,  
																i_pdwResultSet			:= ADR(apExampleLeafModuleInterface), 
																i_udiResultSetSize		:= c_udiMaxExampleLeafModules);
	FOR udiTmp := 1 TO udiCountExampleLeafModules DO
		(* module version check *)
		IF(apExampleLeafModuleInterface[udiTmp]^.q_udiModuleVersion = 1) THEN
			audiExampleLeafModuleId[udiTmp] := apExampleLeafModuleInterface[udiTmp]^.i_udiModuleId;
			asExampleLeafModuleName[udiTmp] := apExampleLeafModuleInterface[udiTmp]^.i_sModuleName;
		END_IF
	END_FOR
	
	q_xReady	:= TRUE;
	
	q_etDiag	:= GD.ET_Diag.Ok;
	q_etDiagExt	:= ET_DiagExtExampleLeafModule.Working;
	q_sMsg		:= '';
	
ELSIF NOT i_xEnable AND xEnableFlag THEN
	xEnableFlag := FALSE;
	
	q_xActive				:= FALSE;	
	q_xReady				:= FALSE;
	q_etDiag				:= GD.ET_Diag.Ok;
	q_etDiagExt				:= ET_DiagExtExampleLeafModule.Disabled;
	q_sMsg					:= '';
	q_udiSetAsCurrentModule	:= 0;		
	q_udiSetAsJogTarget		:= 0;		
END_IF

IF i_xEnable THEN
	q_udiSetAsCurrentModule := udiSetAsCurrentModule;
	udiSetAsCurrentModule := 0;
END_IF


(*********************************************************************)


IF i_xEnable THEN
	IF i_pstCurrentStandardItf = 0 THEN
		q_xReady := FALSE;
		q_etDiag := GD.ET_Diag.InputParameterInvalid;
		q_etDiagExt := ET_DiagExtExampleLeafModule.CurrentStandardItfInvalidPointer;
		q_sMsg := '';
	ELSIF i_dwCurrentAddItf = 0 THEN
		q_xReady := FALSE;
		q_etDiag := GD.ET_Diag.InputParameterInvalid;
		q_etDiagExt := ET_DiagExtExampleLeafModule.CurrentAddItfInvalidPointer;
		q_sMsg := '';
	ELSE
		q_xReady	:= TRUE;
	
		q_etDiag	:= GD.ET_Diag.Ok;
		q_etDiagExt	:= ET_DiagExtExampleLeafModule.Working;
		q_sMsg		:= '';
		
		IF (i_pstCurrentStandardItf^.q_dwModuleType = UDINT_TO_DWORD(ET_ModuleType.ExampleLeafModule)) THEN
			(* Module version check *)
			IF(i_pstCurrentStandardItf^.q_udiModuleVersion = 1) THEN
				pstCurrentExampleLeafModuleInterface := i_dwCurrentAddItf;
				xCurrentIsOfMyType := TRUE;
			END_IF
		ELSE
			pstCurrentExampleLeafModuleInterface := 0;
			xCurrentIsOfMyType := FALSE;
		END_IF	
	
		IF(xCurrentIsOfMyType) THEN
			(* Execute changes requested by user first *)
			IF(NOT xInitUserInputs) THEN
				xInitUserInputs := TRUE;
				(* Ignore values of variables now *)
			ELSE
				(* Detect user changes *)
				IF stCurrentExampleLeafModuleInterface.i_lrPosMax <> lrPosMax THEN
					pstCurrentExampleLeafModuleInterface^.i_lrPosMax := stCurrentExampleLeafModuleInterface.i_lrPosMax;
				END_IF
	
				(* ... *)
			END_IF
			stCurrentExampleLeafModuleInterface := pstCurrentExampleLeafModuleInterface^;
	
		ELSE
			;
			(* Reset other flags *)
		END_IF
	END_IF
ELSE
	xCurrentIsOfMyType := FALSE;
END_IF

END_FUNCTION_BLOCK

// Project Information/GetBooleanProperty
// This function has been automatically generated from the project information.
{attribute 'signature_flag' := '1073741824'}
{attribute 'register_in_runtime'}
FUNCTION GetBooleanProperty : BOOL
VAR_INPUT
	stKey: WSTRING;
END_VAR

IF stKey = "Git:IsGitManaged" THEN
	GetBooleanProperty := FALSE;
ELSIF stKey = "Svn:IsSvnManaged" THEN
	GetBooleanProperty := FALSE;
ELSE
	GetBooleanProperty := FALSE;
END_IF

END_FUNCTION

// Project Information/GetCompany
// This function has been automatically generated from the project information.
{attribute 'signature_flag' := '1073741824'}
{attribute 'register_in_runtime'}
FUNCTION GetCompany : WSTRING
VAR_INPUT
	
END_VAR

GetCompany := "";

END_FUNCTION

// Project Information/GetNumberProperty
// This function has been automatically generated from the project information.
{attribute 'signature_flag' := '1073741824'}
{attribute 'register_in_runtime'}
FUNCTION GetNumberProperty : DINT
VAR_INPUT
	stKey: WSTRING;
END_VAR

GetNumberProperty := 0;

END_FUNCTION

// Project Information/GetTextProperty2
// This function has been automatically generated from the project information.
{attribute 'signature_flag' := '1073741824'}
{attribute 'register_in_runtime'}
FUNCTION GetTextProperty2 : POINTER TO WSTRING
VAR_INPUT
	stKey: WSTRING;
END_VAR

IF stKey = "Author" THEN
	GetTextProperty2 := ADR("SESA697794");
ELSIF stKey = "Company" THEN
	GetTextProperty2 := ADR("");
ELSIF stKey = "DefaultNamespace" THEN
	GetTextProperty2 := ADR("MulticarrierExample ");
ELSIF stKey = "Description" THEN
	GetTextProperty2 := ADR("");
ELSIF stKey = "Project" THEN
	GetTextProperty2 := ADR("Git_example");
ELSIF stKey = "Title" THEN
	GetTextProperty2 := ADR("Git_example");
ELSE
	GetTextProperty2 := ADR("");
END_IF

END_FUNCTION

// Project Information/GetTextProperty
// This function has been automatically generated from the project information.
{attribute 'signature_flag' := '1073741824'}
{attribute 'register_in_runtime'}
FUNCTION GetTextProperty : WSTRING
VAR_INPUT
	stKey: WSTRING;
END_VAR

IF stKey = "Author" THEN
	GetTextProperty := "SESA697794";
ELSIF stKey = "Company" THEN
	GetTextProperty := "";
ELSIF stKey = "DefaultNamespace" THEN
	GetTextProperty := "MulticarrierExample ";
ELSIF stKey = "Description" THEN
	GetTextProperty := "";
ELSIF stKey = "Project" THEN
	GetTextProperty := "Git_example";
ELSIF stKey = "Title" THEN
	GetTextProperty := "Git_example";
ELSE
	GetTextProperty := "";
END_IF

END_FUNCTION

// Project Information/GetTitle
// This function has been automatically generated from the project information.
{attribute 'signature_flag' := '1073741824'}
{attribute 'register_in_runtime'}
FUNCTION GetTitle : WSTRING
VAR_INPUT
	
END_VAR

GetTitle := "Git_example";

END_FUNCTION

// Project Information/GetVersion
// This function has been automatically generated from the project information.
{attribute 'signature_flag' := '1073741824'}
{attribute 'register_in_runtime'}
FUNCTION GetVersion : VERSION
VAR_INPUT
	
END_VAR

GetVersion.uiMajor := 0;
GetVersion.uiMinor := 0;
GetVersion.uiServicePack := 0;
GetVersion.uiPatch := 0;

END_FUNCTION

// Project Information/GetVersionProperty
// This function has been automatically generated from the project information.
{attribute 'signature_flag' := '1073741824'}
{attribute 'register_in_runtime'}
FUNCTION GetVersionProperty : VERSION
VAR_INPUT
	stKey: WSTRING;
END_VAR

IF stKey = "Version" THEN
	GetVersionProperty.uiMajor := 0;
	GetVersionProperty.uiMinor := 0;
	GetVersionProperty.uiServicePack := 0;
	GetVersionProperty.uiPatch := 0;
ELSE
	GetVersionProperty.uiMajor := 0;
	GetVersionProperty.uiMinor := 0;
	GetVersionProperty.uiServicePack := 0;
	GetVersionProperty.uiPatch := 0;
END_IF

END_FUNCTION

// LMC_PacDrive/Application/Check_Lib/CheckBounds
// Implicitly generated code : DO NOT EDIT
FUNCTION CheckBounds : DINT
VAR_INPUT
	index, lower, upper: DINT;
END_VAR

IF  index < lower THEN
	CheckBounds := lower;
	FC_DiagMsgWrite(4, CONCAT('CB min>', CONCAT('idx=', DINT_TO_STRING(index))));
	FC_SysUserCallStack(0);
ELSIF  index > upper THEN
	CheckBounds := upper;
	FC_DiagMsgWrite(4, CONCAT('CB max<', CONCAT('idx=', DINT_TO_STRING(index))));
	FC_SysUserCallStack(0);
ELSE  
	CheckBounds := index;
END_IF

END_FUNCTION

// LMC_PacDrive/Application/Check_Lib/CheckDivDInt
// Implicitly generated code : DO NOT EDIT
FUNCTION CheckDivDInt : DINT
VAR_INPUT
	divisor: DINT;
END_VAR

IF divisor = 0 THEN
	CheckDivDInt:=1;
	FC_DiagMsgWrite(4, 'CDDI Div by 0');
	FC_SysUserCallStack(0);
ELSE
	CheckDivDInt:=divisor;
END_IF

END_FUNCTION

// LMC_PacDrive/Application/Check_Lib/CheckDivLInt
// Implicitly generated code : DO NOT EDIT
FUNCTION CheckDivLInt : LINT
VAR_INPUT
	divisor: LINT;
END_VAR

IF divisor = 0 THEN
	CheckDivLInt:=1;
	FC_DiagMsgWrite(4, 'CDLI Div by 0');
	FC_SysUserCallStack(0);
ELSE
	CheckDivLInt:=divisor;
END_IF

END_FUNCTION

// LMC_PacDrive/Application/Check_Lib/CheckDivLReal
// Implicitly generated code : DO NOT EDIT
FUNCTION CheckDivLReal : LREAL
VAR_INPUT
	divisor: LREAL;
END_VAR

IF divisor = 0 THEN
	CheckDivLReal:=1;
	FC_DiagMsgWrite(4, 'CDLR Div by 0');
	FC_SysUserCallStack(0);
ELSE
	CheckDivLReal:=divisor;
END_IF

END_FUNCTION

// LMC_PacDrive/Application/Check_Lib/CheckDivReal
// Implicitly generated code : DO NOT EDIT
FUNCTION CheckDivReal : REAL
VAR_INPUT
	divisor: REAL;
END_VAR

IF divisor = 0 THEN
	CheckDivReal:=1;
	FC_DiagMsgWrite(4, 'CDR Div by 0');
	FC_SysUserCallStack(0);
ELSE
	CheckDivReal:=divisor;
END_IF

END_FUNCTION

// LMC_PacDrive/Application/Check_Lib/CheckPointer
// Implicitly generated code : DO NOT EDIT
FUNCTION CheckPointer : POINTER TO BYTE
VAR_INPUT
	ptToTest: POINTER TO BYTE; // Destination address of the pointer
	iSize: DINT;            // Size of the type the pointer points to. (e.g: 20 for POINTER TO ARRAY [0..9] OF INT)
	iGran: DINT;		// Granularity of the pointer access. This is the size of the biggest non-structured data type in the type the pointer points to. (e.g: 2 for POINTER TO ARRAY [0..9] OF INT)
	bWrite: BOOL;		// Indicates read or write Access. TRUE = write access.
END_VAR

CheckPointer := ptToTest;
IF ptToTest = 0 THEN
	FC_DiagMsgWrite(4, 'CP = 0');
	FC_SysUserCallStack(0);
ELSE
	CheckPointer := ptToTest;
END_IF

END_FUNCTION

// LMC_PacDrive/Application/Check_Lib/CheckRangeSigned
// Implicitly generated code : DO NOT EDIT
FUNCTION CheckRangeSigned : DINT
VAR_INPUT
	value, lower, upper: DINT;
END_VAR

IF (value < lower) THEN
	CheckRangeSigned := lower;
	FC_DiagMsgWrite(4, CONCAT('CB min>', CONCAT('idx=', DINT_TO_STRING(value))));
	FC_SysUserCallStack(0);
ELSIF(value > upper) THEN
	CheckRangeSigned := upper;
	FC_DiagMsgWrite(4, CONCAT('CB max<', CONCAT('idx=', DINT_TO_STRING(value))));
	FC_SysUserCallStack(0);
ELSE
	CheckRangeSigned := value;
END_IF

END_FUNCTION

// LMC_PacDrive/Application/Check_Lib/CheckRangeUnsigned
// Implicitly generated code : DO NOT EDIT
FUNCTION CheckRangeUnsigned : UDINT
VAR_INPUT
	value, lower, upper: UDINT;
END_VAR

IF (value < lower) THEN
	CheckRangeUnsigned := lower;
	FC_DiagMsgWrite(4, CONCAT('CB min>', CONCAT('idx=', UDINT_TO_STRING(value))));
	FC_SysUserCallStack(0);
ELSIF(value > upper) THEN
	CheckRangeUnsigned := upper;
	FC_DiagMsgWrite(4, CONCAT('CB max<', CONCAT('idx=', UDINT_TO_STRING(value))));
	FC_SysUserCallStack(0);
ELSE
	CheckRangeUnsigned := value;
END_IF

END_FUNCTION

// LMC_PacDrive/Application/TemplateFullProgrammingFramework/EquipmentModules/MulticarrierModule/FC_LrealEqual
FUNCTION FC_LrealEqual : BOOL
VAR_INPUT
	i_lrInput1 : LREAL;
	i_lrInput2 : LREAL;
END_VAR

FC_LrealEqual := ABS(i_lrInput1 - i_lrInput2) < MCR.GCL.Gc_lrCompareTolerance;

END_FUNCTION

// LMC_PacDrive/Application/TemplateFullProgrammingFramework/Examples/ExampleLeafModule/FB_ExampleLeafModule
FUNCTION_BLOCK FB_ExampleLeafModule

VAR_IN_OUT
(* TPL.ST_StandardModuleInterface *)	
	iq_stStandardModuleItf			: TPL.ST_StandardModuleInterface;
	
(* ExceptionHandling and Logging *)	
	iq_stExceptionList				: TPL.ST_ExceptionList;
	iq_stLogDataList				: TPL.ST_LogDataList;
	
(* ST_ExampleLeafModuleInterface *)
	iq_stExampleLeafModuleItf		: ST_ExampleLeafModuleInterface;
END_VAR

VAR
	xEnableFlag : BOOL;
	
	udii : UDINT;
	
	xInitHomingDone : BOOL;
	xNotAbleToSetException : BOOL;

	etDiagBuffer		: GD.ET_Diag;
	etDiagExtBufferTPL	: TPL.ET_DiagExt;
	sDiagMsgBuffer		: STRING[80];
	
	xDiagQuitFlag : BOOL;
	
	
	xExceptionReactionOutsideRange		: BOOL;
	
	stExceptionInit						: TPL.ST_Exception;
	stExceptionCmdImpossibleState		: TPL.ST_Exception;
	stExceptionCmdUnknown				: TPL.ST_Exception;
	stExceptionCmdImpossibleOverwrite	: TPL.ST_Exception;
	stWarningCmdImpossibleReaction		: TPL.ST_Exception;
	stExceptionHoming					: TPL.ST_Exception;
	stExceptionModuleReaction1			: TPL.ST_Exception;
	stExceptionModuleReaction2			: TPL.ST_Exception;
	stExceptionModuleReaction3			: TPL.ST_Exception;
	stExceptionModuleReaction4			: TPL.ST_Exception;
	stExceptionDriveFatal				: TPL.ST_Exception;
	stExcepitonDrive					: TPL.ST_Exception;
	stWarningDrive						: TPL.ST_Exception;

	stModuleReaction			: TPL.ST_Reaction;
	stLocalReaction				: TPL.ST_Reaction;
	stEmptyReaction				: TPL.ST_Reaction;
	stReaction1					: TPL.ST_Reaction;
	stReaction2					: TPL.ST_Reaction;
	stReaction3					: TPL.ST_Reaction;
	stReaction4					: TPL.ST_Reaction;

	udiDoSomethingCounter	: UDINT := 0;

	xCheckCmdException	: BOOL;
	xOpModeCmd			: BOOL;
	xCommandRefused		: BOOL;

	(* OpMode enable and active flags *)
	xHomingEnable : BOOL;
	xHomingActive : BOOL;
	xAutoEnable : BOOL;
	xAutoActive : BOOL;

	xCommandAcceptedInThisCycle : BOOL;

	xHomingException : BOOL;

	xRandomExceptionTrigger: BOOL;

	xStartFlag : BOOL;

	fbLogger : TPL.FB_Logger;
	fbLoggerPoint	: APL.FB_LoggerPoint;
	
	etStateOld : ET_ExampleLeafModuleState;
	udiMyResultSource : UDINT;
	
	ifRefActualValuesPosition : SystemConfigurationItf.IF_RefActualValuesPosition; 
	xSuccess : BOOL;
END_VAR

VAR CONSTANT
	c_udiDoSomeThingLevel : UDINT := 500;
END_VAR

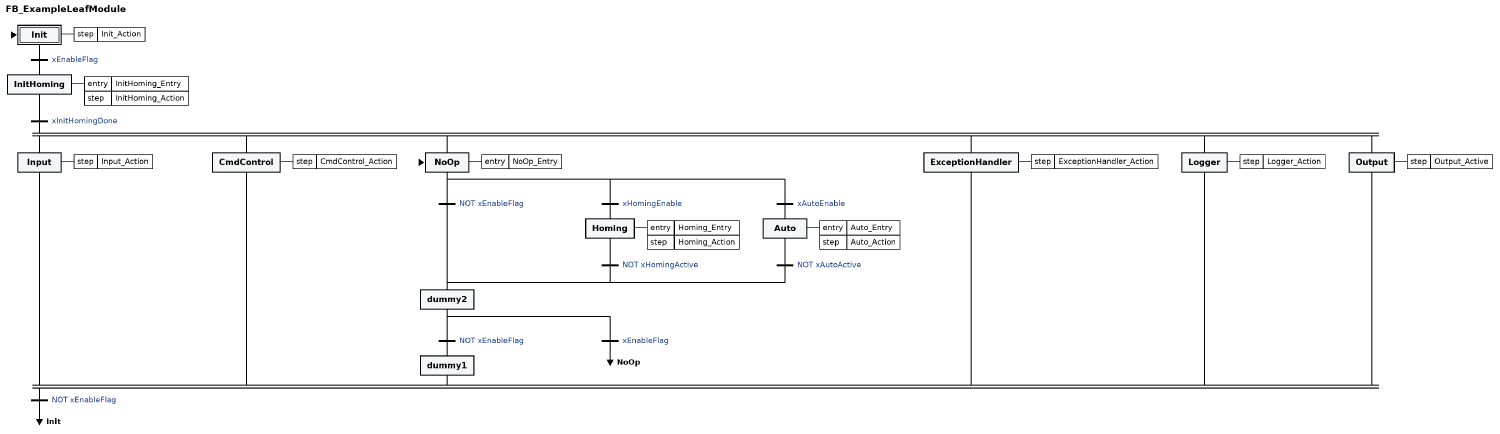
INITIAL_STEP Init:
    Init_Action(N);  // step action
END_STEP
TRANSITION FROM Init TO InitHoming
    := xEnableFlag;
END_TRANSITION
STEP InitHoming:
    InitHoming_Entry(P1);  // entry action
    InitHoming_Action(N);  // step action
END_STEP
TRANSITION FROM InitHoming TO (Input, CmdControl, NoOp, ExceptionHandler, Logger, Output)
    := xInitHomingDone;
END_TRANSITION
STEP Input:
    Input_Action(N);  // step action
END_STEP
STEP CmdControl:
    CmdControl_Action(N);  // step action
END_STEP
STEP NoOp:
    NoOp_Entry(P1);  // entry action
END_STEP
TRANSITION FROM NoOp TO dummy2
    := NOT xEnableFlag;
END_TRANSITION
TRANSITION FROM NoOp TO Homing
    := xHomingEnable;
END_TRANSITION
STEP Homing:
    Homing_Entry(P1);  // entry action
    Homing_Action(N);  // step action
END_STEP
TRANSITION FROM Homing TO dummy2
    := NOT xHomingActive;
END_TRANSITION
TRANSITION FROM NoOp TO Auto
    := xAutoEnable;
END_TRANSITION
STEP Auto:
    Auto_Entry(P1);  // entry action
    Auto_Action(N);  // step action
END_STEP
TRANSITION FROM Auto TO dummy2
    := NOT xAutoActive;
END_TRANSITION
STEP dummy2:
END_STEP
TRANSITION FROM dummy2 TO dummy1
    := NOT xEnableFlag;
END_TRANSITION
TRANSITION FROM dummy2 TO NoOp
    := xEnableFlag;
END_TRANSITION
STEP dummy1:
END_STEP
STEP ExceptionHandler:
    ExceptionHandler_Action(N);  // step action
END_STEP
STEP Logger:
    Logger_Action(N);  // step action
END_STEP
STEP Output:
    Output_Active(N);  // step action
END_STEP
TRANSITION FROM (Input, CmdControl, dummy1, ExceptionHandler, Logger, Output) TO Init
    := NOT xEnableFlag;
END_TRANSITION

ACTION Auto_Action:
(* Start application code *)
IF(iq_stExampleLeafModuleItf.q_etState = ET_ExampleLeafModuleState.AutoWaitForStart) THEN
	IF(xAutoEnable) THEN
		IF(xStartFlag) THEN
			iq_stExampleLeafModuleItf.q_etState := ET_ExampleLeafModuleState.AutoRunning;
		END_IF
	ELSE
		xAutoActive := FALSE;
	END_IF
END_IF

IF(NOT xStartFlag AND iq_stExampleLeafModuleItf.q_etState = ET_ExampleLeafModuleState.AutoRunning) THEN
	iq_stExampleLeafModuleItf.q_etState := ET_ExampleLeafModuleState.AutoWaitForStart;
END_IF

IF(iq_stExampleLeafModuleItf.q_etState = ET_ExampleLeafModuleState.AutoRunning) THEN
	IF(xAutoEnable) THEN
		iq_stExampleLeafModuleItf.q_xValue := ifRefActualValuesPosition.RefPosition >= iq_stExampleLeafModuleItf.i_lrPosMin AND 
													ifRefActualValuesPosition.RefPosition <= iq_stExampleLeafModuleItf.i_lrPosMax;
	ELSE
		iq_stExampleLeafModuleItf.q_etState := ET_ExampleLeafModuleState.AutoWaitForStart;
	END_IF
END_IF
(* End application code *)
END_ACTION

ACTION Auto_Entry:
iq_stExampleLeafModuleItf.q_etState := ET_ExampleLeafModuleState.AutoWaitForStart;
xAutoActive := TRUE;
END_ACTION

METHOD CancelException
VAR_IN_OUT
	iq_stException	: TPL.ST_Exception;
END_VAR
TPL.FC_SetException(	i_xExceptionActive	:= FALSE,
						iq_stException		:= iq_stException,
						iq_stExceptionList	:= iq_stExceptionList,
						iq_stLogDataList	:= iq_stLogDataList,
						q_etDiag 			=> etDiagBuffer,
						q_etDiagExt 		=> etDiagExtBufferTPL,
						q_sMsg 				=> sDiagMsgBuffer);
END_METHOD

ACTION CheckCmd:
(*--------------------------------------------------------------------------------------------------*)
(* CheckCMD is checking if CMD is supported by this module *)
(*--------------------------------------------------------------------------------------------------*)
xOpModeCMD			:= FALSE;
xCheckCmdException	:= FALSE;

IF 	iq_stStandardModuleItf.iq_diCMD = ET_ExampleLeafModuleCmd.Homing OR
	iq_stStandardModuleItf.iq_diCMD = ET_ExampleLeafModuleCmd.Auto OR
	iq_stStandardModuleItf.iq_diCMD = ET_ExampleLeafModuleCmd.Stop THEN

	xOpModeCMD := TRUE;
ELSIF iq_stStandardModuleItf.iq_diCMD = ET_ExampleLeafModuleCmd.Start OR
	  iq_stStandardModuleItf.iq_diCMD = ET_ExampleLeafModuleCmd.Hold THEN
	;
ELSE
	xCheckCmdException := TRUE;
END_IF
END_ACTION

ACTION CmdControl_Action:
(* CMD execution

	algorithm:
	----------

	detect new command?
		check command?
			execute command;
		end
	end

	is command running (at least one cycle)?	
		is command finished?
			signal success/unsuccessful
		end
	end
*)

xCommandAcceptedInThisCycle := FALSE;

(* Detect new command *)
IF(iq_stStandardModuleItf.i_xEnable) THEN
	IF (iq_stStandardModuleItf.iq_diCMD > 0 AND (NOT iq_stStandardModuleItf.q_xCMDActive (* In case no command is active *)
			OR iq_stStandardModuleItf.iq_diCMD <> iq_stStandardModuleItf.q_diCMDActive) (* In case a command is active *)) THEN
	
		xCommandRefused := FALSE; (* Flag is set by RefuseCommand() action *)
	
		(* Check command *)
		CheckCmd();
		IF(xCheckCmdException) THEN
			(*** Check for unknown command ***)
			stExceptionCmdUnknown.sMsg := Standard.CONCAT('Cmd unknown: ',DINT_TO_STRING(iq_stStandardModuleItf.iq_diCmd));
			ReportException(iq_stException := stExceptionCmdUnknown); 
			RefuseCommand();
		ELSE
			(*** Check for impossible overwrite ***)
			IF(iq_stStandardModuleItf.q_xCMDActive AND iq_stStandardModuleItf.iq_diCMD <> ET_ExampleLeafModuleCmd.Stop) THEN (* In this module only the ET_ExampleLeafModuleCmd.Stop command can overwrite other commands *)
				stExceptionCmdImpossibleOverwrite.sMsg := PDL.FC_MultiConcat(	i_sString1 := 'Cmd impossible: ',
																				i_sString2 := FC_EtExampleLeafModuleCmdToString(i_diCmd := iq_stStandardModuleItf.iq_diCmd),
																				i_sString3 := '; Cmd active: ',
																				i_sString4 := FC_EtExampleLeafModuleCmdToString(i_diCmd := iq_stStandardModuleItf.q_diCmdActive) );
				ReportException(iq_stException := stExceptionCmdImpossibleOverwrite);	
				RefuseCommand();
			ELSE
				(*** Check for impossible state ***)
				IF(NOT xOpModeCmd AND (* In this module, all OpMode commands are always possible independent of the state *)
					(iq_stExampleLeafModuleItf.q_etState = ET_ExampleLeafModuleState.NoOp (* Start and Hold are not possible in NoOp *)
					OR (iq_stExampleLeafModuleItf.q_etState = ET_ExampleLeafModuleState.HomingWaitForStart OR iq_stExampleLeafModuleItf.q_etState = ET_ExampleLeafModuleState.HomingDone) AND iq_stStandardModuleItf.iq_diCMD = ET_ExampleLeafModuleCmd.Hold) (* Hold is not supported in homing *)
					) THEN
					stExceptionCmdImpossibleState.sMsg := PDL.FC_MultiConcat(	i_sString1 := 'Cmd impossible: ',
																				i_sString2 := FC_EtExampleLeafModuleCmdToString(i_diCmd := iq_stStandardModuleItf.iq_diCmd),
																				i_sString3 := '; State: ',
																				i_sString4 := FC_EtExampleLeafModuleStateToString(i_etState := iq_stExampleLeafModuleItf.q_etState) );
					ReportException(iq_stException := stExceptionCmdImpossibleState);
					RefuseCommand();
				ELSE
					(* Check for impossible commands due to active error reactions *)
					IF	iq_stStandardModuleItf.iq_diCMD = ET_ExampleLeafModuleCmd.Start 
							AND (stModuleReaction.axReaction[TPL.ET_Reaction.AsyncStop] OR 
								 stModuleReaction.axReaction[TPL.ET_Reaction.SyncStopEH] OR 
								 stModuleReaction.axReaction[TPL.ET_Reaction.SyncStopEL] OR 
								 stModuleReaction.axReaction[TPL.ET_Reaction.StopEndOfCycle]) (* Start impossible if error reaction 4 or higher *)
						OR 
						
						iq_stStandardModuleItf.iq_diCMD <> ET_ExampleLeafModuleCmd.Stop 
							AND (stModuleReaction.axReaction[TPL.ET_Reaction.AsyncStop] OR 
								 stModuleReaction.axReaction[TPL.ET_Reaction.SyncStopEH] OR 
								 stModuleReaction.axReaction[TPL.ET_Reaction.SyncStopEL]) THEN (* Everything else, with exception of Stop, impossible if error reaction 3 or higher *)

						stWarningCmdImpossibleReaction.sMsg := PDL.FC_MultiConcat(	i_sString1 := 'Cmd impossible: ',
																					i_sString2 := FC_EtExampleLeafModuleCmdToString(i_diCmd := iq_stStandardModuleItf.iq_diCmd),
																					i_sString3 := '; Reaction: ',
																					i_sString4 := TPL.FC_GetStandardReactionName(iq_stReaction := stModuleReaction));
						ReportException(iq_stException := stWarningCmdImpossibleReaction);
						RefuseCommand();
					END_IF
				END_IF
			END_IF
		END_IF
	
		IF(NOT xCommandRefused) THEN (* Command has passed all checks, execute command *)
			IF fbLoggerPoint.etLogLevel >= APL.ET_LogLevel.UserAction THEN
				fbLoggerPoint.AddLogEntry(	i_etLogLevel	:= APL.ET_LogLevel.UserAction,
											i_etDiag		:= GD.ET_Diag.Ok,
											i_udiDiagExt	:= ET_DiagExtExampleLeafModule.Ok,
											i_sMessage		:= Standard.CONCAT(Standard.CONCAT(Standard.CONCAT('Command executing: ', FC_etExampleLeafModuleCmdToString(i_diCmd := iq_stStandardModuleItf.iq_diCmd)),' number: '),DINT_TO_STRING(iq_stStandardModuleItf.iq_diCmd)),
											q_etDiag		:= ,
											q_etDiagExt		:= );
			END_IF
			(* Accept command *)
			iq_stStandardModuleItf.q_xCMDActive := TRUE;
			iq_stStandardModuleItf.q_xCMDDone := FALSE;
			iq_stStandardModuleItf.q_diCMDActive := iq_stStandardModuleItf.iq_diCMD;
	
			xCommandAcceptedInThisCycle := TRUE; (* Signal for command done checks *)
	
			IF(xOpModeCMD) THEN
				DisableAllJobs();
				
				CASE iq_stStandardModuleItf.iq_diCMD OF
					ET_ExampleLeafModuleCmd.Stop:
						;	(* Do nothing, disabled OpMode flags automatically lead to NoOp *)
						
					ET_ExampleLeafModuleCmd.Homing:
						xHomingEnable := TRUE;
					
					ET_ExampleLeafModuleCmd.Auto:
						xAutoEnable := TRUE;
				END_CASE
			ELSE
				(* Action commands *)
				CASE iq_stStandardModuleItf.iq_diCMD OF
					ET_ExampleLeafModuleCmd.Start:
						xStartFlag := TRUE;
					
					ET_ExampleLeafModuleCmd.Hold:
						xStartFlag := FALSE;
				END_CASE
			END_IF
		END_IF (* New command? *)
	END_IF

(********************************************* Check successful and unsucessful of given commands ****************************************)

	(* Check if active command is done or is stopped by an error *)
	IF(NOT xCommandAcceptedInThisCycle) THEN (* Don't execute these checks if we accepted a new command in this cycle
		to ensure that execution of every command requires a minimum of 2 cycles *)

		IF(iq_stStandardModuleItf.q_xCMDActive) THEN
			CASE iq_stStandardModuleItf.iq_diCmd OF
				ET_ExampleLeafModuleCmd.Homing:
					(* Successful *)
					IF(xHomingActive) THEN
						SignalSuccessfulExecution();
					END_IF
					(* Unsucessful *)
					IF (stModuleReaction.axReaction[TPL.ET_Reaction.AsyncStop] OR 
						stModuleReaction.axReaction[TPL.ET_Reaction.SyncStopEL] OR 
						stModuleReaction.axReaction[TPL.ET_Reaction.SyncStopEH]) THEN
						
						SignalUnsuccessfulExecution();
					END_IF
					
				ET_ExampleLeafModuleCmd.Auto:
					(* Successful *)
					IF(xAutoActive) THEN
						SignalSuccessfulExecution();
					END_IF
					(* Unsucessful *)
					IF (stModuleReaction.axReaction[TPL.ET_Reaction.AsyncStop] OR 
						stModuleReaction.axReaction[TPL.ET_Reaction.SyncStopEL] OR 
						stModuleReaction.axReaction[TPL.ET_Reaction.SyncStopEH]) THEN

						SignalUnsuccessfulExecution();
					END_IF
	
				ET_ExampleLeafModuleCmd.Stop:
					(* Successful *)
					IF(iq_stExampleLeafModuleItf.q_etState = ET_ExampleLeafModuleState.NoOp) THEN
						SignalSuccessfulExecution();
					END_IF
					
				ET_ExampleLeafModuleCmd.Start:
					IF(iq_stExampleLeafModuleItf.q_etState = ET_ExampleLeafModuleState.HomingDone) THEN
						xStartFlag := FALSE;
					END_IF
					(* Successful *)
					IF(iq_stExampleLeafModuleItf.q_etState = ET_ExampleLeafModuleState.HomingDone AND NOT xHomingException
						OR iq_stExampleLeafModuleItf.q_etState = ET_ExampleLeafModuleState.AutoRunning) THEN
						SignalSuccessfulExecution();
					END_IF
					(* Unsucessful *)
					IF (stModuleReaction.axReaction[TPL.ET_Reaction.AsyncStop] OR 
						stModuleReaction.axReaction[TPL.ET_Reaction.SyncStopEL] OR 
						stModuleReaction.axReaction[TPL.ET_Reaction.SyncStopEH] OR 
						stModuleReaction.axReaction[TPL.ET_Reaction.StopEndOfCycle]  OR
						iq_stExampleLeafModuleItf.q_etState = ET_ExampleLeafModuleState.HomingDone AND xHomingException) THEN
						
						SignalUnsuccessfulExecution();
					END_IF
					
				ET_ExampleLeafModuleCmd.Hold:
					(* Successful *)
					IF(iq_stExampleLeafModuleItf.q_etState = ET_ExampleLeafModuleState.AutoWaitForStart) THEN
						SignalSuccessfulExecution();
					END_IF
					(* Unsucessful *)
					IF (stModuleReaction.axReaction[TPL.ET_Reaction.AsyncStop] OR 
						stModuleReaction.axReaction[TPL.ET_Reaction.SyncStopEL] OR 
						stModuleReaction.axReaction[TPL.ET_Reaction.SyncStopEH]) THEN

						SignalUnsuccessfulExecution();
					END_IF
			END_CASE
		END_IF
	END_IF
ELSE
	(* Module is going to be disabled *)
	iq_stStandardModuleItf.q_xReady := FALSE;
	xEnableFlag := FALSE;
	
	DisableAllJobs();
	
	xStartFlag := FALSE;

	IF(iq_stStandardModuleItf.q_xCmdActive) THEN (* If a command is currently active, cancel its execution *)
		SignalUnsuccessfulExecution();
	ELSE
		InactiveCmdExecution(); (* Command processing as if we were disabled *)
	END_IF
END_IF
END_ACTION

ACTION DiagQuit:
IF(iq_stStandardModuleItf.i_xDiagQuit AND NOT xDiagQuitFlag) THEN
	(* Rising edge of error quit *)
	xDiagQuitFlag := TRUE;
	xNotAbleToSetException := FALSE;

	FOR udii := 1 TO TPL.ET_Reaction.MainsContactorOff DO
		stLocalReaction.axReaction[udii] := FALSE;
	END_FOR

	iq_stStandardModuleItf.q_etDiag := GD.ET_Diag.Ok;

	IF(iq_stStandardModuleItf.iq_diCMD < 0) THEN
		iq_stStandardModuleItf.iq_diCMD := 0;
	END_IF
	IF fbLoggerPoint.etLogLevel >= APL.ET_LogLevel.UserAction THEN
		fbLoggerPoint.AddLogEntry(	i_etLogLevel	:= APL.ET_LogLevel.UserAction,
									i_etDiag		:= GD.ET_Diag.Ok,
									i_udiDiagExt	:= ET_DiagExtExampleLeafModule.Ok,
									i_sMessage		:= 'Diag Quit',
									q_etDiag		:= ,
									q_etDiagExt		:= );
	END_IF
ELSIF(NOT iq_stStandardModuleItf.i_xDiagQuit AND xDiagQuitFlag) THEN
	xDiagQuitFlag := FALSE;
END_IF
END_ACTION

ACTION DisableAllJobs:
(* Disable current OpMode and enable next one *)
xHomingEnable := FALSE;
xAutoEnable := FALSE;

xStartFlag := FALSE; (* On OpMode change, always reset the start flag *)
END_ACTION

ACTION ExceptionHandler_Action:
(* -----------------------------------------------------------------------------------------------*)
(* Check Axis Errors *)
(* -----------------------------------------------------------------------------------------------*)
	IF (iq_stExampleLeafModuleItf.i_ifDrive.DiagClass > 3) THEN
		stExceptionDriveFatal.sMsg := PDL.FC_MultiConcat(	i_sString1 := 'DiagCode: ',
															i_sString2 := DINT_TO_STRING(iq_stExampleLeafModuleItf.i_ifDrive.DiagCode),
															i_sString3 := ' Msg: ',
															i_sString4 := iq_stExampleLeafModuleItf.i_ifDrive.DiagMsg);
															
		ReportException(iq_stException := stExceptionDriveFatal);
		
	ELSIF (iq_stExampleLeafModuleItf.i_ifDrive.DiagClass = 3) THEN
		stExcepitonDrive.sMsg := PDL.FC_MultiConcat(	i_sString1 := 'DiagCode: ',
														i_sString2 := DINT_TO_STRING(iq_stExampleLeafModuleItf.i_ifDrive.DiagCode),
														i_sString3 := ' Msg: ',
														i_sString4 := iq_stExampleLeafModuleItf.i_ifDrive.DiagMsg);
														
		ReportException(iq_stException := stExcepitonDrive);
		
	ELSIF (iq_stExampleLeafModuleItf.i_ifDrive.DiagClass > 0)  AND (iq_stExampleLeafModuleItf.i_ifDrive.DiagClass < 3) THEN
		stWarningDrive.sMsg := PDL.FC_MultiConcat(	i_sString1 := 'DiagCode: ',
													i_sString2 := DINT_TO_STRING(iq_stExampleLeafModuleItf.i_ifDrive.DiagCode),
													i_sString3 := ' Msg: ',
													i_sString4 := iq_stExampleLeafModuleItf.i_ifDrive.DiagMsg);
													
		ReportException(iq_stException := stWarningDrive);
	END_IF

(* -----------------------------------------------------------------------------------------------*)
(* Check StopModi *)
(* -----------------------------------------------------------------------------------------------*)
IF (NOT iq_stStandardModuleItf.i_xEnable OR 
	stModuleReaction.axReaction[TPL.ET_Reaction.AsyncStop] OR 
	stModuleReaction.axReaction[TPL.ET_Reaction.SyncStopEL] OR 
	stModuleReaction.axReaction[TPL.ET_Reaction.SyncStopEH]) THEN

	xAutoEnable := FALSE;
	xHomingEnable := FALSE;
END_IF
IF (NOT iq_stStandardModuleItf.i_xEnable OR 
	stModuleReaction.axReaction[TPL.ET_Reaction.AsyncStop] OR 
	stModuleReaction.axReaction[TPL.ET_Reaction.SyncStopEL] OR 
	stModuleReaction.axReaction[TPL.ET_Reaction.SyncStopEH] OR 
	stModuleReaction.axReaction[TPL.ET_Reaction.StopEndOfCycle] ) THEN

	xStartFlag := FALSE;
END_IF
END_ACTION

ACTION Homing_Action:
(* Start application code *)
IF(xStartFlag AND (iq_stExampleLeafModuleItf.q_etState = ET_ExampleLeafModuleState.HomingWaitForStart OR iq_stExampleLeafModuleItf.q_etState = ET_ExampleLeafModuleState.HomingDone)) THEN
	xHomingException := FALSE;
	iq_stExampleLeafModuleItf.q_etState := ET_ExampleLeafModuleState.HomingExecuting;
END_IF

IF(iq_stExampleLeafModuleItf.q_etState = ET_ExampleLeafModuleState.HomingExecuting) THEN
	(* Emulating an action in the process that takes some time *)
	udiDoSomethingCounter := udiDoSomethingCounter + 1;
	IF(udiDoSomethingCounter > c_udiDoSomeThingLevel) THEN
		(* Homing done *)
		iq_stExampleLeafModuleItf.q_xValue := TRUE;

		(* Sometimes creates an error *)
		IF(iq_stExampleLeafModuleItf.i_xEnableRandomExceptionTrigger) THEN
			IF(xRandomExceptionTrigger) THEN
				xHomingException := TRUE;
			END_IF
			xRandomExceptionTrigger := NOT xRandomExceptionTrigger;
		END_IF

		iq_stExampleLeafModuleItf.q_etState := ET_ExampleLeafModuleState.HomingDone;
	END_IF
END_IF

IF xHomingException THEN
	ReportException(iq_stException := stExceptionHoming);
ELSE
	CancelException(iq_stException := stExceptionHoming);
END_IF

IF(iq_stExampleLeafModuleItf.q_etState <> ET_ExampleLeafModuleState.HomingExecuting) THEN
	(* If homing is not running, allow exit of homing by xHomingEnable = FALSE *)
	IF(NOT xHomingEnable) THEN
		xHomingActive := FALSE;
	END_IF
END_IF
(* End application code *)
END_ACTION

ACTION Homing_Entry:
iq_stExampleLeafModuleItf.q_etState := ET_ExampleLeafModuleState.HomingWaitForStart;
xHomingActive := TRUE;


(* Start application code *)
udiDoSomethingCounter := 0;
(* End application code *)
END_ACTION

ACTION InactiveCmdExecution:
(* Command execution if module is not active (q_xActive = FALSE) or currently deactivating (i_xEnable = FALSE, q_xActive is still TRUE) *)
IF iq_stStandardModuleItf.iq_diCmd <> 0 THEN
	IF(NOT iq_stStandardModuleItf.i_xEnable) THEN
		iq_stStandardModuleItf.iq_diCmd := 0; (* All commands are signaled executed if module is disabled *)
(*ELSE*)
	ELSIF(iq_stStandardModuleItf.iq_diCmd > 0) THEN (* New command *)
		(* Command execution during enable but module is not ready for commands yet ==> error *)
		//xExceptionCmdImpossibleState := TRUE;

		stExceptionCmdImpossibleState.sMsg := PDL.FC_MultiConcat(	i_sString1 := 'Cmd impossible: ',
																	i_sString2 := FC_EtExampleLeafModuleCmdToString(i_diCmd := ABS(iq_stStandardModuleItf.iq_diCmd)),
																	i_sString3 := '; State: ',
																	i_sString4 := FC_EtExampleLeafModuleStateToString(i_etState := iq_stExampleLeafModuleItf.q_etState));
		ReportException(iq_stException := stExceptionCmdImpossibleState);
		iq_stStandardModuleItf.iq_diCmd:= - ABS(iq_stStandardModuleItf.iq_diCmd);
	END_IF
END_IF
iq_stStandardModuleItf.q_xCmdActive := FALSE;
iq_stStandardModuleItf.q_xCmdDone := FALSE;
iq_stStandardModuleItf.q_diCmdActive := 0;
END_ACTION

ACTION Init_Action:
iq_stStandardModuleItf.q_xActive			:= FALSE;
iq_stStandardModuleItf.q_xReady				:= FALSE;

iq_stStandardModuleItf.q_etDiag				:= GD.ET_Diag.Ok;
iq_stStandardModuleItf.q_udiDiagExt			:= ET_DiagExtExampleLeafModule.Disabled;
iq_stStandardModuleItf.q_sDiagExt			:= FC_EtDiagExtExampleLeafModuleToString(i_etDiagExt := iq_stStandardModuleItf.q_udiDiagExt);
iq_stStandardModuleItf.q_sMsg				:= '';

iq_stStandardModuleItf.q_dwModuleType		:= ET_ModuleType.ExampleLeafModule;
iq_stStandardModuleItf.q_sModuleTypeName	:= 'ExampleLeafModule';
iq_stStandardModuleItf.q_udiModuleVersion	:= 1;

iq_stExampleLeafModuleItf.q_etState	:= ET_ExampleLeafModuleState.Disabled;

THIS^.DiagQuit();
THIS^.InactiveCmdExecution();

udiMyResultSource := ET_ExceptionSource.ExampleLeafModule; (* Has to be coded this way to get around compiler restrictions*)

(* detect invalid configurations and avoid array index out of range error *)
IF(iq_stStandardModuleItf.iq_stExt.udiReactionOffset + TPL. ET_Reaction.MainsContactorOff > TPL.Gc_udiMaxNumberOfReactions) OR xExceptionReactionOutsideRange THEN (* module uses error reactions 1 to 5 *)
	xExceptionReactionOutsideRange := TRUE; (* create unquittable error *)
	
	(* create exception *)
	stExceptionInit.etDiag					:= GD.ET_Diag.InputParameterInvalid;
	stExceptionInit.udiDiagExt				:= ET_DiagExtExampleLeafModule.ReactionOffsetRange;
	stExceptionInit.sMsg					:= Standard.CONCAT('Value: ', UDINT_TO_STRING(iq_stStandardModuleItf.iq_stExt.udiReactionOffset));
	stExceptionInit.udiModuleId				:= iq_stStandardModuleItf.i_udiModuleId;
	stExceptionInit.sModuleName				:= iq_stStandardModuleItf.i_sModuleName;
	stExceptionInit.etSource				:= udiMyResultSource;
	stExceptionInit.timDelayTime			:= T#0MS;
	stExceptionInit.wHmiAttributes			:= 0;
	stExceptionInit.xAutoQuit				:= FALSE;
	stExceptionInit.stReaction.axReaction[TPL.ET_Reaction.AsyncStop]	:= TRUE; (* without offset on purpose *)
	
	iq_stStandardModuleItf.iq_stExt.udiReactionOffset := 0;
	
	ReportException(iq_stException := stExceptionInit);
ELSIF (iq_stStandardModuleItf.i_xEnable) THEN
	stReaction1 := stEmptyReaction;
	stReaction1.axReaction[iq_stStandardModuleItf.iq_stExt.udiReactionOffset + TPL.ET_Reaction.AsyncStop] := TRUE;
	stReaction2 := stEmptyReaction;
	stReaction2.axReaction[iq_stStandardModuleItf.iq_stExt.udiReactionOffset + TPL.ET_Reaction.SyncStopEL] := TRUE;
	stReaction3 := stEmptyReaction;
	stReaction3.axReaction[iq_stStandardModuleItf.iq_stExt.udiReactionOffset + TPL.ET_Reaction.SyncStopEH] := TRUE;
	stReaction4 := stEmptyReaction;
	stReaction4.axReaction[iq_stStandardModuleItf.iq_stExt.udiReactionOffset + TPL.ET_Reaction.StopEndOfCycle] := TRUE;
	
	(* Initialization of exception structures *)
	stExceptionCmdUnknown.etDiag						:= GD.ET_Diag.ExecutionAborted;
	stExceptionCmdUnknown.udiDiagExt					:= ET_DiagExtExampleLeafModule.CmdUnknown;
	stExceptionCmdUnknown.sMsg							:= 'Command unknown'; (* Replaced on usage *)
	stExceptionCmdUnknown.udiModuleId					:= iq_stStandardModuleItf.i_udiModuleId;
	stExceptionCmdUnknown.sModuleName					:= iq_stStandardModuleItf.i_sModuleName;
	stExceptionCmdUnknown.etSource						:= udiMyResultSource;
	stExceptionCmdUnknown.timDelayTime					:= T#0MS;
	stExceptionCmdUnknown.wHmiAttributes				:= 0;
	stExceptionCmdUnknown.xAutoQuit						:= FALSE;
	stExceptionCmdUnknown.stReaction					:= stReaction1;

	stExceptionCmdImpossibleOverwrite.etDiag			:= GD.ET_Diag.ExecutionAborted;
	stExceptionCmdImpossibleOverwrite.udiDiagExt		:= ET_DiagExtExampleLeafModule.CmdImpossibleOverwrite;
	stExceptionCmdImpossibleOverwrite.sMsg				:= 'Impossible command overwrite'; (* Replaced on usage *)
	stExceptionCmdImpossibleOverwrite.udiModuleId		:= iq_stStandardModuleItf.i_udiModuleId;
	stExceptionCmdImpossibleOverwrite.sModuleName		:= iq_stStandardModuleItf.i_sModuleName;
	stExceptionCmdImpossibleOverwrite.etSource			:= udiMyResultSource;
	stExceptionCmdImpossibleOverwrite.timDelayTime		:= T#0MS;
	stExceptionCmdImpossibleOverwrite.wHmiAttributes	:= 0;
	stExceptionCmdImpossibleOverwrite.xAutoQuit			:= FALSE;
	stExceptionCmdImpossibleOverwrite.stReaction		:= stReaction1;
	
	stExceptionCmdImpossibleState.etDiag				:= GD.ET_Diag.ExecutionAborted;
	stExceptionCmdImpossibleState.udiDiagExt			:= ET_DiagExtExampleLeafModule.CmdImpossibleState;
	stExceptionCmdImpossibleState.sMsg					:= 'Impossible command for state'; (* Replaced on usage *)
	stExceptionCmdImpossibleState.udiModuleId			:= iq_stStandardModuleItf.i_udiModuleId;
	stExceptionCmdImpossibleState.sModuleName			:= iq_stStandardModuleItf.i_sModuleName;
	stExceptionCmdImpossibleState.etSource				:= udiMyResultSource;
	stExceptionCmdImpossibleState.timDelayTime			:= T#0MS;
	stExceptionCmdImpossibleState.wHmiAttributes		:= 0;
	stExceptionCmdImpossibleState.xAutoQuit				:= FALSE;
	stExceptionCmdImpossibleState.stReaction			:= stReaction1;

	stWarningCmdImpossibleReaction.etDiag				:= GD.ET_Diag.ExecutionAborted;
	stWarningCmdImpossibleReaction.udiDiagExt			:= ET_DiagExtExampleLeafModule.CmdImpossibleReaction;
	stWarningCmdImpossibleReaction.sMsg					:= 'Impossible command on reaction'; (* Replaced on usage *)
	stWarningCmdImpossibleReaction.udiModuleId			:= iq_stStandardModuleItf.i_udiModuleId;
	stWarningCmdImpossibleReaction.sModuleName			:= iq_stStandardModuleItf.i_sModuleName;
	stWarningCmdImpossibleReaction.etSource				:= udiMyResultSource;
	stWarningCmdImpossibleReaction.timDelayTime			:= T#0MS;
	stWarningCmdImpossibleReaction.wHmiAttributes		:= 0;
	stWarningCmdImpossibleReaction.xAutoQuit			:= FALSE;
	
	stExceptionModuleReaction1.etDiag					:= GD.ET_Diag.InputParameterInvalid;(* Replaced on usage *)
	stExceptionModuleReaction1.udiDiagExt				:= ET_DiagExtExampleLeafModule.Ok;(* Replaced on usage *)
	stExceptionModuleReaction1.sMsg						:= '';(* Replaced on usage *)
	stExceptionModuleReaction1.udiModuleId				:= iq_stStandardModuleItf.i_udiModuleId;
	stExceptionModuleReaction1.sModuleName				:= iq_stStandardModuleItf.i_sModuleName;
	stExceptionModuleReaction1.etSource					:= udiMyResultSource;
	stExceptionModuleReaction1.timDelayTime				:= T#0MS;
	stExceptionModuleReaction1.wHmiAttributes			:= 0;
	stExceptionModuleReaction1.xAutoQuit				:= FALSE;
	stExceptionModuleReaction1.stReaction				:= stReaction1;

	stExceptionModuleReaction2.etDiag					:= GD.ET_Diag.InputParameterInvalid;(* Replaced on usage *)
	stExceptionModuleReaction2.udiDiagExt				:= ET_DiagExtExampleLeafModule.Ok;(* Replaced on usage *)
	stExceptionModuleReaction2.sMsg						:= '';(* Replaced on usage *)
	stExceptionModuleReaction2.udiModuleId				:= iq_stStandardModuleItf.i_udiModuleId;
	stExceptionModuleReaction2.sModuleName				:= iq_stStandardModuleItf.i_sModuleName;
	stExceptionModuleReaction2.etSource					:= udiMyResultSource;
	stExceptionModuleReaction2.timDelayTime				:= T#0MS;
	stExceptionModuleReaction2.wHmiAttributes			:= 0;
	stExceptionModuleReaction2.xAutoQuit				:= FALSE;
	stExceptionModuleReaction2.stReaction				:= stReaction2;

	stExceptionModuleReaction3.etDiag					:= GD.ET_Diag.InputParameterInvalid;(* Replaced on usage *)
	stExceptionModuleReaction3.udiDiagExt				:= ET_DiagExtExampleLeafModule.Ok;(* Replaced on usage *)
	stExceptionModuleReaction3.sMsg						:= '';(* Replaced on usage *)
	stExceptionModuleReaction3.udiModuleId				:= iq_stStandardModuleItf.i_udiModuleId;
	stExceptionModuleReaction3.sModuleName				:= iq_stStandardModuleItf.i_sModuleName;
	stExceptionModuleReaction3.etSource					:= udiMyResultSource;
	stExceptionModuleReaction3.timDelayTime				:= T#0MS;
	stExceptionModuleReaction3.wHmiAttributes			:= 0;
	stExceptionModuleReaction3.xAutoQuit				:= FALSE;
	stExceptionModuleReaction3.stReaction				:= stReaction3;

	stExceptionModuleReaction4.etDiag					:= GD.ET_Diag.InputParameterInvalid;(* Replaced on usage *)
	stExceptionModuleReaction4.udiDiagExt				:= ET_DiagExtExampleLeafModule.Ok;(* Replaced on usage *)
	stExceptionModuleReaction4.sMsg						:= '';(* Replaced on usage *)
	stExceptionModuleReaction4.udiModuleId				:= iq_stStandardModuleItf.i_udiModuleId;
	stExceptionModuleReaction4.sModuleName				:= iq_stStandardModuleItf.i_sModuleName;
	stExceptionModuleReaction4.etSource					:= udiMyResultSource;
	stExceptionModuleReaction4.timDelayTime				:= T#0MS;
	stExceptionModuleReaction4.wHmiAttributes			:= 0;
	stExceptionModuleReaction4.xAutoQuit				:= FALSE;
	stExceptionModuleReaction4.stReaction				:= stReaction4;
	
	stExceptionDriveFatal.etDiag						:= GD.ET_Diag.DriveConditionInvalid;
	stExceptionDriveFatal.udiDiagExt					:= ET_DiagExtExampleLeafModule.DriveFatalException;
	stExceptionDriveFatal.sMsg							:= 'Drive diag'; (* Replaced on usage *)
	stExceptionDriveFatal.udiModuleId					:= iq_stStandardModuleItf.i_udiModuleId;
	stExceptionDriveFatal.sModuleName					:= iq_stStandardModuleItf.i_sModuleName;
	stExceptionDriveFatal.etSource						:= udiMyResultSource;
	stExceptionDriveFatal.timDelayTime					:= T#0MS;
	stExceptionDriveFatal.wHmiAttributes				:= 0;
	stExceptionDriveFatal.xAutoQuit						:= FALSE;
	stExceptionDriveFatal.stReaction					:= stReaction1;
	
	stExcepitonDrive.etDiag								:= GD.ET_Diag.DriveConditionInvalid;
	stExcepitonDrive.udiDiagExt							:= ET_DiagExtExampleLeafModule.DriveException;
	stExcepitonDrive.sMsg								:= 'Drive diag'; (* Replaced on usage *)
	stExcepitonDrive.udiModuleId						:= iq_stStandardModuleItf.i_udiModuleId;
	stExcepitonDrive.sModuleName						:= iq_stStandardModuleItf.i_sModuleName;
	stExcepitonDrive.etSource							:= udiMyResultSource;
	stExcepitonDrive.timDelayTime						:= T#0MS;
	stExcepitonDrive.wHmiAttributes						:= 0;
	stExcepitonDrive.xAutoQuit							:= FALSE;
	stExcepitonDrive.stReaction							:= stReaction2;

	stWarningDrive.etDiag								:= GD.ET_Diag.DriveConditionInvalid;
	stWarningDrive.udiDiagExt							:= ET_DiagExtExampleLeafModule.DriveWarning;
	stWarningDrive.sMsg									:= 'Drive warning'; (* Replaced on usage *)
	stWarningDrive.udiModuleId							:= iq_stStandardModuleItf.i_udiModuleId;
	stWarningDrive.sModuleName							:= iq_stStandardModuleItf.i_sModuleName;
	stWarningDrive.etSource								:= udiMyResultSource;
	stWarningDrive.timDelayTime							:= T#0MS;
	stWarningDrive.wHmiAttributes						:= 0;
	stWarningDrive.xAutoQuit							:= FALSE;
	stWarningDrive.stReaction							:= stReaction4;

	stExceptionInit.etDiag								:= GD.ET_Diag.InputParameterInvalid; (* Replaced on usage *)
	stExceptionInit.udiDiagExt							:= ET_DiagExtExampleLeafModule.Ok; (* Replaced on usage *)
	stExceptionInit.sMsg								:= ''; (* Replaced on usage *)
	stExceptionInit.udiModuleId							:= iq_stStandardModuleItf.i_udiModuleId;
	stExceptionInit.sModuleName							:= iq_stStandardModuleItf.i_sModuleName;
	stExceptionInit.etSource							:= udiMyResultSource;
	stExceptionInit.timDelayTime						:= T#0MS;
	stExceptionInit.wHmiAttributes						:= 0;
	stExceptionInit.xAutoQuit							:= FALSE;
	stExceptionInit.stReaction							:= stReaction1;
	
	stExceptionHoming.etDiag							:= GD.ET_Diag.HomingFailed;
	stExceptionHoming.udiDiagExt						:= ET_DiagExtExampleLeafModule.RandomException;
	stExceptionHoming.sMsg								:= '';
	stExceptionHoming.udiModuleId						:= iq_stStandardModuleItf.i_udiModuleId;
	stExceptionHoming.sModuleName						:= iq_stStandardModuleItf.i_sModuleName;
	stExceptionHoming.etSource							:= udiMyResultSource;
	stExceptionHoming.timDelayTime						:= T#0MS;
	stExceptionHoming.wHmiAttributes					:= 0;
	stExceptionHoming.xAutoQuit							:= FALSE;
	stExceptionHoming.stReaction						:= stReaction4;

	IF (iq_stExampleLeafModuleItf.i_ifDrive = 0) THEN
		stExceptionModuleReaction1.etDiag		:= GD.ET_Diag.InputParameterInvalid;
		stExceptionModuleReaction1.udiDiagExt	:= ET_DiagExtExampleLeafModule.DriveInvalid;
		stExceptionModuleReaction1.sMsg			:= 'No drive given';
		
		ReportException(iq_stException := stExceptionModuleReaction1);
	ELSE
		xEnableFlag := TRUE;
		iq_stStandardModuleItf.q_xActive := TRUE;
		
		FOR udii := 1 TO TPL.Gc_udiMaxNumberOfReactions DO
			stLocalReaction.axReaction[udii] := FALSE;
		END_FOR
		
		THIS^.SetInterfaces();
		
		xInitHomingDone := FALSE;
		
		iq_stExampleLeafModuleItf.q_etState := ET_ExampleLeafModuleState.Initializing;
		
		iq_stStandardModuleItf.q_etDiag		:= GD.ET_Diag.Ok;
		iq_stStandardModuleItf.q_udiDiagExt	:= ET_DiagExtExampleLeafModule.Initializing;
		iq_stStandardModuleItf.q_sDiagExt	:= FC_EtDiagExtExampleLeafModuleToString(ET_DiagExtExampleLeafModule.Initializing);
		iq_stStandardModuleItf.q_sMsg		:= '';
		
		IF fbLoggerPoint.etLogLevel >= APL.ET_LogLevel.UserAction THEN
			fbLoggerPoint.AddLogEntry(	i_etLogLevel	:= APL.ET_LogLevel.UserAction,
										i_etDiag		:= GD.ET_Diag.Ok,
										i_udiDiagExt	:= ET_DiagExtExampleLeafModule.Ok,
										i_sMessage		:= 'enabeling Module',
										q_etDiag		:= ,
										q_etDiagExt		:= );
		END_IF
	END_IF

END_IF

THIS^.SetOutputs();
END_ACTION

ACTION InitHoming_Action:
DiagQuit();
InactiveCmdExecution();

(* Emulating an initialization that takes some time *)
udiDoSomethingCounter := udiDoSomethingCounter + 1;
IF(iq_stExampleLeafModuleItf.i_xInitHoming) THEN
	xInitHomingDone := FALSE;
	iq_stExampleLeafModuleItf.q_xValue := TRUE;
	IF(udiDoSomethingCounter > c_udiDoSomeThingLevel) THEN
		(* Initial homing done *)
		xInitHomingDone := TRUE;
		iq_stExampleLeafModuleItf.q_xValue := TRUE;
		IF fbLoggerPoint.etLogLevel >= APL.ET_LogLevel.StatusMessage THEN
			fbLoggerPoint.AddLogEntry(	i_etLogLevel	:= APL.ET_LogLevel.StatusMessage,
										i_etDiag		:= GD.ET_Diag.Ok,
										i_udiDiagExt	:= ET_DiagExtExampleLeafModule.Ok,
										i_sMessage		:= 'InitHoming done',
										q_etDiag		:= ,
										q_etDiagExt		:= );
		END_IF
	END_IF
ELSE
	xInitHomingDone := TRUE;
END_IF

THIS^.SetOutputs();
END_ACTION

ACTION InitHoming_Entry:
udiDoSomethingCounter := 0;
END_ACTION

ACTION Input_Action:
iq_stStandardModuleItf.q_xReady := TRUE;
THIS^.DiagQuit();

(* -----------------------------------------------------------------------------------------------*)
(* Check external Reaction *)
(* -----------------------------------------------------------------------------------------------*)
stModuleReaction.axReaction[TPL.ET_Reaction.AsyncStop] := stLocalReaction.axReaction[TPL.ET_Reaction.AsyncStop] OR iq_stStandardModuleItf.i_stReaction.axReaction[TPL.ET_Reaction.AsyncStop];
stModuleReaction.axReaction[TPL.ET_Reaction.SyncStopEL] := stLocalReaction.axReaction[TPL.ET_Reaction.SyncStopEL] OR iq_stStandardModuleItf.i_stReaction.axReaction[TPL.ET_Reaction.SyncStopEL];
stModuleReaction.axReaction[TPL.ET_Reaction.SyncStopEH] := stLocalReaction.axReaction[TPL.ET_Reaction.SyncStopEH] OR iq_stStandardModuleItf.i_stReaction.axReaction[TPL.ET_Reaction.SyncStopEH];
stModuleReaction.axReaction[TPL.ET_Reaction.StopEndOfCycle] := stLocalReaction.axReaction[TPL.ET_Reaction.StopEndOfCycle] OR iq_stStandardModuleItf.i_stReaction.axReaction[TPL.ET_Reaction.StopEndOfCycle];
stModuleReaction.axReaction[TPL.ET_Reaction.MainsContactorOff] := stLocalReaction.axReaction[TPL.ET_Reaction.MainsContactorOff] OR iq_stStandardModuleItf.i_stReaction.axReaction[TPL.ET_Reaction.MainsContactorOff];
END_ACTION

ACTION Logger_Action:
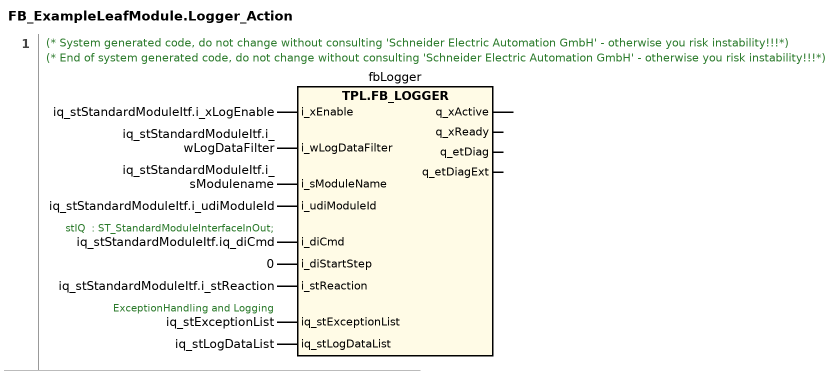
// NETWORK 1
// 					(* System generated code, do not change without consulting 'Schneider Electric Automation GmbH' - otherwise you risk instability!!!*)
// (* End of system generated code, do not change without consulting 'Schneider Electric Automation GmbH' - otherwise you risk instability!!!*)
//
//   iq_stStandardModuleItf.iq_diCmd: stIQ : ST_StandardModuleInterfaceInOut;
//   iq_stExceptionList: ExceptionHandling and Logging
fbLogger(
    i_xEnable := iq_stStandardModuleItf.i_xLogEnable,
    i_wLogDataFilter := iq_stStandardModuleItf.i_wLogDataFilter,
    i_sModuleName := iq_stStandardModuleItf.i_sModulename,
    i_udiModuleId := iq_stStandardModuleItf.i_udiModuleId,
    i_diCmd := iq_stStandardModuleItf.iq_diCmd,
    i_diStartStep := 0,
    i_stReaction := iq_stStandardModuleItf.i_stReaction,
    iq_stExceptionList := iq_stExceptionList,
    iq_stLogDataList := iq_stLogDataList); // TPL.FB_LOGGER
END_ACTION

ACTION NoOp_Entry:
iq_stExampleLeafModuleItf.q_etState := ET_ExampleLeafModuleState.NoOp;
END_ACTION

ACTION Output_Active:
(* System generated code, to be changed by experienced programmers *)
THIS^.SetOutputs();
(* End of system generated code, to be changed by experienced programmers *)
END_ACTION

ACTION RefuseCommand:
iq_stStandardModuleItf.q_xCMDActive := FALSE;
iq_stStandardModuleItf.q_xCMDDone := FALSE;
iq_stStandardModuleItf.iq_diCMD := - iq_stStandardModuleItf.iq_diCMD;

xCommandRefused := TRUE;
END_ACTION

METHOD PUBLIC RegisterLoggerPoint
VAR_INPUT
	i_ifParent		: APL.IF_LoggerPoint;
	i_sName			: STRING[80];
END_VAR
VAR_OUTPUT
	q_etDiag		: GD.ET_Diag := GD.ET_Diag.Ok;
	q_etDiagExt		: ET_DiagExtExampleLeafModule := ET_DiagExtExampleLeafModule.Ok;
	q_sMsg			: STRING[80] := '';
END_VAR
VAR
	etDiagBuffer		: GD.ET_Diag;
	etDiagExtBufferAPL	: APL.ET_DiagExt;
END_VAR
THIS^.fbLoggerPoint.RegisterLoggerPoint(	i_ifParent		:= i_ifParent,
											i_sName			:= i_sName,
											i_sType			:= 'FB_ExampleLeafModule',
											i_sSource		:= 'Project',
											q_etDiag		=> etDiagBuffer,
											q_etDiagExt		=> etDiagExtBufferAPL);
IF (etDiagBuffer <> GD.ET_Diag.Ok) THEN
	CASE etDiagExtBufferAPL OF
		APL.ET_DiagExt.ParentInvalid:
			q_etDiag := GD.ET_Diag.InputParameterInvalid;
			q_etDiagExt := ET_DiagExtExampleLeafModule.ParentInvalid;
			
		APL.ET_DiagExt.ParentNotRegistered:
			q_etDiag := GD.ET_Diag.InputParameterInvalid;
			q_etDiagExt := ET_DiagExtExampleLeafModule.ParentNotRegistered;
			
		APL.ET_DiagExt.MaxNumberOfLoggerPointsExeeded:
			q_etDiag := GD.ET_Diag.InputParameterInvalid;
			q_etDiagExt := ET_DiagExtExampleLeafModule.MaxNumberOfLoggerPointsExeeded;
			
	ELSE
		q_etDiag := GD.ET_Diag.UnexpectedProgramBehavior;
		q_etdiagExt := ET_DiagExtExampleLeafModule.UnexpectedDiagExt;
		q_sMsg := Standard.CONCAT('RegisterLoggerPoint: ', APL.FC_EtDiagExtToString(i_etDiagExt := etDiagExtBufferAPL));
	END_CASE
END_IF
END_METHOD

METHOD ReportException
VAR_IN_OUT
	iq_stException	: TPL.ST_Exception;
END_VAR
VAR CONSTANT
	c_diMaxReaction	: DINT := 4;
END_VAR
IF (fbLoggerPoint.etLogLevel >= APL.ET_LogLevel.CriticalException) AND (iq_stException.etDiag = GD.ET_Diag.UnexpectedProgramBehavior) THEN
	IF NOT TPL.FC_CheckExceptionIsInList( iq_stException := iq_stException, iq_stExceptionList := THIS^.iq_stExceptionList) THEN
		fbLoggerPoint.AddLogEntry(	i_etLogLevel	:= APL.ET_LogLevel.CriticalException,
									i_etDiag		:= GD.ET_Diag.Ok,
									i_udiDiagExt	:= ET_DiagExtExampleLeafModule.Ok,
									i_sMessage		:= Standard.CONCAT(Standard.CONCAT(Standard.CONCAT(Standard.CONCAT(Standard.CONCAT(Standard.CONCAT('Exception ET_Diag: ',GD.FC_EtDiagToString(i_etDiag := iq_stException.etDiag)),' ET_DiagExt: '),FC_EtDiagExtToString(i_etDiagExt := iq_stException.udiDiagExt)),' sMsg: '),iq_stException.sMsg),TPL.FC_GetStandardReactionName(iq_stReaction := iq_stException.stReaction)),
									q_etDiag		:= ,
									q_etDiagExt		:= );
	END_IF
ELSIF (fbLoggerPoint.etLogLevel >= APL.ET_LogLevel.Exception) THEN
	IF NOT TPL.FC_CheckExceptionIsInList( iq_stException := iq_stException, iq_stExceptionList := THIS^.iq_stExceptionList) THEN
		fbLoggerPoint.AddLogEntry(	i_etLogLevel	:= APL.ET_LogLevel.Exception,
									i_etDiag		:= GD.ET_Diag.Ok,
									i_udiDiagExt	:= ET_DiagExtExampleLeafModule.Ok,
									i_sMessage		:= Standard.CONCAT(Standard.CONCAT(Standard.CONCAT(Standard.CONCAT(Standard.CONCAT(Standard.CONCAT('Exception ET_Diag: ',GD.FC_EtDiagToString(i_etDiag := iq_stException.etDiag)),' ET_DiagExt: '),FC_EtDiagExtToString(i_etDiagExt := iq_stException.udiDiagExt)),' sMsg: '),iq_stException.sMsg),TPL.FC_GetStandardReactionName(iq_stReaction := iq_stException.stReaction)),
									q_etDiag		:= ,
									q_etDiagExt		:= );
	END_IF
END_IF

iq_stException.sDiagExt := FC_EtDiagExtExampleLeafModuleToString(i_etDiagExt := iq_stException.udiDiagExt);
TPL.FC_SetException(	i_xExceptionActive	:= TRUE,
						iq_stException		:= iq_stException,
						iq_stExceptionList	:= iq_stExceptionList,
						iq_stLogDataList	:= iq_stLogDataList,
						q_etDiag 			=> etDiagBuffer,
						q_etDiagExt 		=> etDiagExtBufferTPL,
						q_sMsg 				=> sDiagMsgBuffer);
						
IF (etDiagBuffer <> GD.ET_Diag.Ok) THEN
	(* if exception could not be reported, show exception on outputs *)
	xNotAbleToSetException := TRUE;
	iq_stStandardModuleItf.q_etDiag := iq_stException.etDiag;
	iq_stStandardModuleItf.q_udiDiagExt := iq_stException.udiDiagExt;
	iq_stStandardModuleItf.q_sDiagExt := iq_stException.sDiagExt;
	iq_stStandardModuleItf.q_sMsg := iq_stException.sMsg;
END_IF

stLocalReaction.axReaction[TPL.ET_Reaction.MainsContactorOff] := stLocalReaction.axReaction[TPL.ET_Reaction.MainsContactorOff] OR iq_stException.stReaction.axReaction[TPL.ET_Reaction.MainsContactorOff];
stLocalReaction.axReaction[TPL.ET_Reaction.AsyncStop] := stLocalReaction.axReaction[TPL.ET_Reaction.AsyncStop] OR iq_stException.stReaction.axReaction[TPL.ET_Reaction.AsyncStop];
stLocalReaction.axReaction[TPL.ET_Reaction.SyncStopEH] := stLocalReaction.axReaction[TPL.ET_Reaction.SyncStopEH] OR iq_stException.stReaction.axReaction[TPL.ET_Reaction.SyncStopEH];
stLocalReaction.axReaction[TPL.ET_Reaction.SyncStopEL] := stLocalReaction.axReaction[TPL.ET_Reaction.SyncStopEL] OR iq_stException.stReaction.axReaction[TPL.ET_Reaction.SyncStopEL];
(* special handling for StopEndOfCycle. Wait till reaction feedback from machine. User can transform this reaction and make own reaction.
stLocalReaction.axReaction[TPL.ET_Reaction.StopEndOfCycle] := stLocalReaction.axReaction[TPL.ET_Reaction.StopEndOfCycle] OR iq_stException.stReaction.axReaction[TPL.ET_Reaction.StopEndOfCycle];
*)

stModuleReaction.axReaction[TPL.ET_Reaction.MainsContactorOff] := stLocalReaction.axReaction[TPL.ET_Reaction.MainsContactorOff] OR stModuleReaction.axReaction[TPL.ET_Reaction.MainsContactorOff];
stModuleReaction.axReaction[TPL.ET_Reaction.AsyncStop] := stLocalReaction.axReaction[TPL.ET_Reaction.AsyncStop] OR stModuleReaction.axReaction[TPL.ET_Reaction.AsyncStop];
stModuleReaction.axReaction[TPL.ET_Reaction.SyncStopEH] := stLocalReaction.axReaction[TPL.ET_Reaction.SyncStopEH] OR stModuleReaction.axReaction[TPL.ET_Reaction.SyncStopEH];
stModuleReaction.axReaction[TPL.ET_Reaction.SyncStopEL] := stLocalReaction.axReaction[TPL.ET_Reaction.SyncStopEL] OR stModuleReaction.axReaction[TPL.ET_Reaction.SyncStopEL];
(* special handling for StopEndOfCycle. Wait till reaction feedback from machine. User can transform this reaction and make own reaction.
stModuleReaction.axReaction[TPL.ET_Reaction.StopEndOfCycle] := stLocalReaction.axReaction[TPL.ET_Reaction.StopEndOfCycle] OR stModuleReaction.axReaction[TPL.ET_Reaction.StopEndOfCycle];
*)
END_METHOD

METHOD SetInterfaces
VAR_INPUT
END_VAR
IF NOT SYSTEMINTERFACE.FC_IsStLogicalAddressValid(i_stLogAddr := iq_stExampleLeafModuleItf.i_ifDrive.stLogicalAddress) THEN
	stExceptionModuleReaction1.etDiag		:= GD.ET_Diag.InputParameterInvalid;
	stExceptionModuleReaction1.udiDiagExt	:= ET_DiagExtExampleLeafModule.DriveInvalid;
	stExceptionModuleReaction1.sMsg			:= 'i_ifDrive - Invalid logical address.';
	
	ReportException(iq_stException := stExceptionModuleReaction1);
END_IF

